(* CODESYS project CORE.library
   Company: Ziga Javornik
   DefaultNamespace: ZigaLibs.Core
   Version: 0.0.3.7
   Placeholder: ZigaLibs.Core
   Author: Ziga Javornik
   Description: A collection of core objects for work with further libraries implementations.
   Title: ZigaLibs.Core

Project tree, tasks and I/O mapping:
  libraries: Base Interfaces, * (System); Tc2_EtherCAT, * (Beckhoff Automation GmbH); Tc2_IoFunctions, 3.4.5.0 (Beckhoff Automation GmbH); Tc2_Standard, * (Beckhoff Automation GmbH); Tc2_System, * (Beckhoff Automation GmbH); Tc2_Utilities, * (Beckhoff Automation GmbH); Tc3_Module, * (Beckhoff Automation GmbH); TcError, 0.2.2.1 (Roald87); TcUnit, * (www.tcunit.org)
  GVLs/
  SOURCE/
    Array/
      DUTs/
        data type ST_ArrayProperties
        data type T_ArrayIndexer
      program ArrayHelper [ST]: Clear, DoesArrayContainItem, FindLastOccupiedItem, GetElementCount, GetMaxIndex, InsertAtStart, SetAtFirstEmptySlot, ShiftDown, ShiftUp, ValidateArrayVar
    Beckhoff/
      Ads/
        program AdsHelper [ST]: GetEthercatMasterIdFromNetIdString, NetIdToString
        function block FB_HasAmsAddressFromProcessImage [ST]: AmsAddress
        interface I_HasAmsAddress: AmsAddress
      EtherCAT/
        CoE/
          DUTs/
            data type ST_CoeEntry
            data type ST_CoeEntry_DINT
            data type ST_CoeEntry_INT
            data type ST_CoeEntry_REAL
            data type ST_CoeEntry_SINT
            data type ST_CoeEntry_String128
            data type ST_CoeEntry_String255
            data type ST_CoeEntry_String30
            data type ST_CoeEntry_UDINT
            data type ST_CoeEntry_UINT
            data type ST_CoeEntry_USINT
            data type T_CoEIndex
            data type T_CoESubIndex
          function block FB_CoeReadWrite [ST]: ReadAny, WriteAny
          interface I_ReadsCoE: ReadCoE
        Diagnosis/
          DUTs/
            Device state/
              data type E_EcDeviceState
              data type E_EcDeviceStateExtras
              data type E_EcLinkState
              data type ST_EcDeviceState
              data type ST_EcSlaveState
            data type E_EthercatDiagnosisState
            data type E_EthercatDiagnosisStatus
            data type ST_EthercatSlaveInfo
          interface I_EthercatDiagnosis: Error, IgnoredSlaves, IgnoreSlave, MissingSlaves, Reset, Scan, Status
        program EthercatHelper [ST]: ConvertBeckhoffEcStateToCustomStruct, GetBoxNameByAddress
        function block FB_ReadBoxName [ST]
    Errors/
      DUTs/
        data type ST_AdsError
        data type ST_Error
        data type ST_GenericError
      function block FB_ErrorSource [ST]: AdsError, Error, GenericError, ResetError
      interface I_ErrorSource
      interface I_HasAdsError: AdsError
      interface I_HasError: Error
      interface I_HasGenericError: GenericError
    General/
      Memory/
        data type E_MemCmpResults
        function block FB_Malloc [ST]: FB_exit, FB_init, ValidateAction, ValidateIndex, ValidateInputVar, IsAllocated, Properties, Allocate, AllocateAny, Expand, Free, Get, GetPtr, Remove, Set
        program MemoryHelper [ST]: GetRouterStatusInfo
        data type ST_AllocatedMemoryProperties
      Variable extensions/
        function block BoolEx [ST]: HasBeenFalseForAtLeast, HasBeenTrueForAtLeast, HasFallingEdge, HasRisingEdge, IsVarValid, PulseWithInterval, Reset, Set, Toggle, Value
      Variable information/
        function F_DoesVarTypeEqual [ST]
        function F_GetVarInfo [ST]
        data type ST_VarInfo
        data type T_VarInfo
        data type T_VarSize
      function block FB_BooleanObserver [ST]
      function block FB_HasInstanceNameAndPath [ST]: FB_init, InstanceName, InstancePath
      function block FB_HasTaskInfo [ST]: TaskInfo
      function block FB_Watchdog [ST]
      program InstanceNameHelper [ST]: InstanceNameFromPath, RemoveProjectFromInstancePath
      data type ST_Value
    String/
      StringBuilder/
        Extensions/
          AddAny/
            data type E_AddAnyBitOptions
            interface I_StringBuilderEx_Any: AddAny, AddAnyBit, AddAnyReal
        function block FB_StringBuilder [ST]: AddAny, AddAnyBit, AddAnyReal, AddString, AddWithDblQuotationMarks, AddWithQuotationMark, Create, Reset
        interface I_StringBuilder: AddString, AddWithDblQuotationMarks, AddWithQuotationMark, Create, Reset
      program StringConstants [ST]
      program StringHelper [ST]: EndsWith, FindStringWithin, Join, StartsWith, ToLowerCase, ToLowerCase_UnlimitedSize, ToUpperCase, ToUpperCase_UnlimitedSize, TrimLeftSide, TrimRightSide
      data type T_Char
    Time/
      DUTs/
        data type E_TimeFormat
        data type ST_CurrentSystemTimeInfo
      function block FB_DateTimeToStringConverter [ST]: DateTime, Day, Hour, Millisecond, Minute, Month, Second, Year
      function block FB_LocalSystemTimeProvider [ST]: ConvertToString, CurrentTime, SetSystemTime
      interface I_DateTimeToStringConverter: DateTime, Day, Hour, Millisecond, Minute, Month, Second, Year
      interface I_LocalSystemTimeProvider: ConvertToString, CurrentTime
  TESTS/
    Test suites/
      Time/
        function block FB_LocalSystemTime_Tests [ST]: Test01_CheckSystemTime_ExpectValue, Test02_SetSystemTime_ExpectNoErrorAndCorrectTimeRead
      function block FB_AdsHelper_Tests [ST]: Test_MasterAddress, Test_NetIdToString_AllZeros_ExpectEmptyString
      function block FB_ArrayHelper_Tests [ST]: Test01_GetArrayElementCount, Test02_GetArrayMaxIndex, Test03_InsertNumber, Test04_InsertString, Test05_InsertStruct, Test06_ShiftUp_ExpectLastElementOverwriteFirstElementZero, Test07_SetAtFirstEmptySlot, Test08_AllMethods_provideNonArrayVar_ExpectNothing, Test09_InsertIntoEmptyArray_ExpectOnlyFirstItem, Test10_CheckIfArrayContainsItem, Test11_ClearArray_ExpectEmptyArray, Test12_ReferenceToArrayWithAllMethods_ExpectNormalResults, Test13_FindLastOccupiedItem, Test14_ShiftDown_ExpectFirstElementOverwriteLastElementZero
      function block FB_BoolEx_Tests [ST]: Test01_BooleanTrue_ExpectTrueAfterElapsedTime, Test02_BooleanFalse_ExpectTrueAfterElapsedTime, Test03_RisingAndFallingEdge_ExpectPulses, Test04_GetAndSetValue, Test05_Toggle_ExpectValueInverts, Test06_PulseWithInterval_100ms_ExpectValueChangeEvery100ms, Test07_Set_ExpectTrue, Test08_Reset_ExpectFalse
      function block FB_DateTimeToStringConverter_Tests [ST]: Test01_Year, Test02_Month, Test03_Day, Test04_Hour, Test05_Minute, Test06_Second, Test07_Millisecond
      function block FB_ErrorSource_ExtensionForTests [ST]
      function block FB_ErrorSource_Tests [ST]: Test01_ErrorProperty, Test02_ErrorCode, Test03_ErrorMessage, Test04_GenericError
      function block FB_EthercatHelper_Tests [ST]: Test01_ConvertBeckhoffEcState_ProvideAllOptions_ExpectCorrectResults
      function block FB_HasInstanceName_ExtensionForTests [ST]
      function block FB_HasInstanceName_Tests [ST]: Test01_InstanceName, Test02_InstancePath
      function block FB_HasTaskInfo_ExtensionsForTests [ST]
      function block FB_HasTaskInfo_Tests [ST]: Test01_TaskInfoPropertyValidity
      function block FB_Malloc_Tests [ST]: BeforeTestFinish, BeforeTestStart, ValidatePropertiesAfterFailedAllocation, Test01_ProvideIncorrectParameters_ExpectNoAllocation, Test02_Allocate10Integers_ExpectNoError_ValidateProperties, Test03_Free_ExpectNoMemoryAllocated, Test04_SetAndGet_ExpectGetReturnsCorrectValue, Test05_SetAtIncorrectIndex_ExpectFalseReturned, Test06_GetFromIncorrectIndex_ExpectTargetValueUnchanged_MethodReturnFalse, Test07_Expand_ExpectOldDataStillExists_LastDataSetIsEmpty, Test08_Remove_ExpectDataSetToCollapseBy1
      function block FB_StringBuilder_Tests [ST]: Test01_AddStrings_ExpectConcat, Test02_AddWithSingleQuotationMarks, Test03_AddWithDoubleQuotationMarks, Test04_CreateDoesNotResetStringSequence, Test05_ResetClearsBuildSequence
      function block FB_StringBuilderEx_Any_Tests [ST]: Test01_BOOL, Test02_BYTE, Test03_DATE, Test04_DateAndTime, Test05_DINT, Test06_DWORD, Test07_ENUM, Test08_INT, Test09_LINT, Test10_LREAL, Test11_LTIME, Test12_LWORD, Test13_REAL, Test14_SINT, Test15_STRING, Test16_TIME, Test17_TOD, Test18_UDINT, Test19_UINT, Test20_ULINT, Test21_USINT, Test22_WORD, Test23_WSTRING, Test24_ANY_BIT_WORD, Test25_ANY_BIT_BYTE, Test26_ANY_BIT_DWORD, Test27_ANY_BIT_LWORD, Test28_ANY_REAL_REAL, Test29_ANY_REAL_LREAL
      function block FB_StringHelper_Tests [ST]: Test01_StartsWith, Test02_Join, Test03_EndsWith, Test05_Contains, Test06_ToLowerCase_UnlimitedSize, Test07_ToUpperCase_UnlimitedSize
    program PRG_TESTS [ST]
*)

// SOURCE/Array/DUTs/ST_ArrayProperties
TYPE ST_ArrayProperties :
STRUCT
	Count		: DINT;
	StartIndex	: T_ArrayIndexer;
	EndIndex	: T_ArrayIndexer;
END_STRUCT
END_TYPE

// SOURCE/Array/DUTs/T_ArrayIndexer
// Should be used when accessing array index.
TYPE T_ArrayIndexer : DINT; END_TYPE

// SOURCE/Beckhoff/EtherCAT/CoE/DUTs/ST_CoeEntry
{attribute 'qualified_only'}
// CoE entry in the dictionary, includes index and the subindex
TYPE ST_CoeEntry :
STRUCT
	Index		: T_CoEIndex;
	Subindex	: T_CoESubIndex;
END_STRUCT
END_TYPE

// SOURCE/Beckhoff/EtherCAT/CoE/DUTs/ST_CoeEntry_DINT
TYPE ST_CoeEntry_DINT EXTENDS ST_CoeEntry :
STRUCT
	Value	: DINT;
END_STRUCT
END_TYPE

// SOURCE/Beckhoff/EtherCAT/CoE/DUTs/ST_CoeEntry_INT
TYPE ST_CoeEntry_INT EXTENDS ST_CoeEntry :
STRUCT
	Value	: INT;
END_STRUCT
END_TYPE

// SOURCE/Beckhoff/EtherCAT/CoE/DUTs/ST_CoeEntry_REAL
TYPE ST_CoeEntry_REAL EXTENDS ST_CoeEntry :
STRUCT
	Value	: REAL;
END_STRUCT
END_TYPE

// SOURCE/Beckhoff/EtherCAT/CoE/DUTs/ST_CoeEntry_SINT
TYPE ST_CoeEntry_SINT EXTENDS ST_CoeEntry :
STRUCT
	Value	: SINT;
END_STRUCT
END_TYPE

// SOURCE/Beckhoff/EtherCAT/CoE/DUTs/ST_CoeEntry_String128
TYPE ST_CoeEntry_String128 EXTENDS ST_CoeEntry :
STRUCT
	Value	: STRING(128);
END_STRUCT
END_TYPE

// SOURCE/Beckhoff/EtherCAT/CoE/DUTs/ST_CoeEntry_String255
TYPE ST_CoeEntry_String255 EXTENDS ST_CoeEntry :
STRUCT
	Value	: Tc2_System.T_MaxString;
END_STRUCT
END_TYPE

// SOURCE/Beckhoff/EtherCAT/CoE/DUTs/ST_CoeEntry_String30
TYPE ST_CoeEntry_String30 EXTENDS ST_CoeEntry :
STRUCT
	Value	: STRING(30);
END_STRUCT
END_TYPE

// SOURCE/Beckhoff/EtherCAT/CoE/DUTs/ST_CoeEntry_UDINT
TYPE ST_CoeEntry_UDINT EXTENDS ST_CoeEntry :
STRUCT
	Value	: UDINT;
END_STRUCT
END_TYPE

// SOURCE/Beckhoff/EtherCAT/CoE/DUTs/ST_CoeEntry_UINT
TYPE ST_CoeEntry_UINT EXTENDS ST_CoeEntry :
STRUCT
	Value	: UINT;
END_STRUCT
END_TYPE

// SOURCE/Beckhoff/EtherCAT/CoE/DUTs/ST_CoeEntry_USINT
TYPE ST_CoeEntry_USINT EXTENDS ST_CoeEntry :
STRUCT
	Value	: USINT;
END_STRUCT
END_TYPE

// SOURCE/Beckhoff/EtherCAT/CoE/DUTs/T_CoEIndex
TYPE T_CoEIndex : WORD; END_TYPE

// SOURCE/Beckhoff/EtherCAT/CoE/DUTs/T_CoESubIndex
TYPE T_CoESubIndex : BYTE; END_TYPE

// SOURCE/Beckhoff/EtherCAT/Diagnosis/DUTs/Device state/E_EcDeviceState
{attribute 'qualified_only'}
TYPE E_EcDeviceState :
(
	INIT		:= Tc2_EtherCAT.EC_DEVICE_STATE_INIT,
	PREOP		:= Tc2_EtherCAT.EC_DEVICE_STATE_PREOP,
	BOOTSTRAP	:= Tc2_EtherCAT.EC_DEVICE_STATE_BOOTSTRAP,
	SAFEOP		:= Tc2_EtherCAT.EC_DEVICE_STATE_SAFEOP,
	OP			:= Tc2_EtherCAT.EC_DEVICE_STATE_OP
)BYTE;
END_TYPE

// SOURCE/Beckhoff/EtherCAT/Diagnosis/DUTs/Device state/E_EcDeviceStateExtras
{attribute 'qualified_only'}
TYPE E_EcDeviceStateExtras :
(
	NOTHING				:= 16#00,
	STATE_MACHINE_ERROR := Tc2_EtherCAT.EC_DEVICE_STATE_ERROR,
	INVALID_VPRS		:= Tc2_EtherCAT.EC_DEVICE_STATE_INVALID_VPRS,
	INIIT_CMD_ERROR		:= Tc2_EtherCAT.EC_DEVICE_STATE_INITCMD_ERROR,
	DISABLED			:= Tc2_EtherCAT.EC_DEVICE_STATE_DISABLED
)BYTE;
END_TYPE

// SOURCE/Beckhoff/EtherCAT/Diagnosis/DUTs/Device state/E_EcLinkState
TYPE E_EcLinkState :
(
	OK					:= Tc2_EtherCAT.EC_LINK_STATE_OK,
	NOT_PRESENT			:= Tc2_EtherCAT.EC_LINK_STATE_NOT_PRESENT,
	LINK_WITHOUT_COMM	:= Tc2_EtherCAT.EC_LINK_STATE_LINK_WITHOUT_COMM,
	MISSING_LINK		:= Tc2_EtherCAT.EC_LINK_STATE_MISSING_LINK,
	ADDITIONAL_LINK		:= Tc2_EtherCAT.EC_LINK_STATE_ADDITIONAL_LINK,
	PORT_A				:= Tc2_EtherCAT.EC_LINK_STATE_PORT_A,
	PORT_B				:= Tc2_EtherCAT.EC_LINK_STATE_PORT_B,
	PORT_C				:= Tc2_EtherCAT.EC_LINK_STATE_PORT_C,
	PORT_D				:= Tc2_EtherCAT.EC_LINK_STATE_PORT_D
)BYTE;
END_TYPE

// SOURCE/Beckhoff/EtherCAT/Diagnosis/DUTs/Device state/ST_EcDeviceState
TYPE ST_EcDeviceState :
STRUCT
	State		: E_EcDeviceState;	// Device state
	StateExtras	: E_EcDeviceStateExtras;	// Extra information
END_STRUCT
END_TYPE

// SOURCE/Beckhoff/EtherCAT/Diagnosis/DUTs/Device state/ST_EcSlaveState
TYPE ST_EcSlaveState :
STRUCT
	Device	: ST_EcDeviceState;	// Device state
	Link	: E_EcLinkState;	// Link state
END_STRUCT
END_TYPE

// SOURCE/Beckhoff/EtherCAT/Diagnosis/DUTs/E_EthercatDiagnosisState
{attribute 'qualified_only'}
{attribute 'strict'}
TYPE E_EthercatDiagnosisState :
(
	READY,
	GET_SLAVE_STATES,
	GET_FAULTY_SLAVE_ADDRESSES,
	FINISHED,
	ERROR
);
END_TYPE

// SOURCE/Beckhoff/EtherCAT/Diagnosis/DUTs/E_EthercatDiagnosisStatus
TYPE E_EthercatDiagnosisStatus :
(
	NO_ERROR,				// No error, all slaves are present
	MISSING_ALLOWED_SLAVES,	// Missing slaves, but they are allowed (for example, hot connect)
	ERROR					// Missing slaves that are not allowed to be missing
);
END_TYPE

// SOURCE/Beckhoff/EtherCAT/Diagnosis/DUTs/ST_EthercatSlaveInfo
TYPE ST_EthercatSlaveInfo :
STRUCT
	Name		: Tc2_System.T_MaxString;	// Slave name
	IsIgnored	: BOOL;	// True if slave is ignored with the scan
	State		: ST_EcSlaveState;
END_STRUCT
END_TYPE

// SOURCE/Errors/DUTs/ST_AdsError
TYPE ST_AdsError EXTENDS ST_Error:
STRUCT
	Code	: TcError.AdsErrorCodes;
	Message	: Tc2_System.T_MaxString;
END_STRUCT
END_TYPE

// SOURCE/Errors/DUTs/ST_Error
TYPE ST_Error :
STRUCT
	Source	: Tc2_System.T_MaxString;
END_STRUCT
END_TYPE

// SOURCE/Errors/DUTs/ST_GenericError
TYPE ST_GenericError EXTENDS ST_Error :
STRUCT
	Code	: DINT;
	Message	: Tc2_System.T_MaxString;
END_STRUCT
END_TYPE

// SOURCE/General/Memory/E_MemCmpResults
{attribute 'qualified_only'}
TYPE E_MemCmpResults :
(
	pBUFF1_LESS_THAN_pBUFF2	:= -1,
	IDENTICAL	:= 0,
	PbUFF1_GREATER_THAN_pBUFF2	:= 1,
	ERROR	:= 255
)DINT;
END_TYPE

// SOURCE/General/Memory/ST_AllocatedMemoryProperties
// Properties for working with dynamic memory allocation.
TYPE ST_AllocatedMemoryProperties :
STRUCT
	Size				: DINT;		// Size of the allocated memory
	StartAddress		: PVOID;	// Pointer to the address of the array memory space
	BaseTypeSize		: DINT;		// Size of the base type provided, when allocated
	NumberOfElements	: DINT;	// Number of elements provided, when allocated.
END_STRUCT
END_TYPE

// SOURCE/General/Variable information/ST_VarInfo
TYPE ST_VarInfo :
STRUCT
	DataType	: __SYSTEM.TYPE_CLASS;
	Address		: POINTER TO BYTE;
	Size		: T_VarSize;
END_STRUCT
END_TYPE

// SOURCE/General/Variable information/T_VarInfo
TYPE T_VarInfo : __SYSTEM.VAR_INFO; END_TYPE

// SOURCE/General/Variable information/T_VarSize
// Variable size alias type. To be used when working with SIZEOF operator.
TYPE T_VarSize : UXINT; END_TYPE

// SOURCE/General/ST_Value
TYPE ST_Value :
STRUCT
	Setpoint	: REAL;
	Actual		: REAL;
END_STRUCT
END_TYPE

// SOURCE/String/StringBuilder/Extensions/AddAny/E_AddAnyBitOptions
{attribute 'qualified_only'}
{attribute 'strict'}
// Provides various options of how ANY_BIT data type can be converted.
TYPE E_AddAnyBitOptions :
(
	BINARY,			// Will be converted to a binary string (base 2)
	DECIMAL,		// Will be converted to a decial string (base 10)
	HEXADECIMAL,	// Will be converted to hexadecimal string (base 16)
	OCTAL			// Will be converted to octal string (base 8)
);
END_TYPE

// SOURCE/String/T_Char
TYPE T_Char : STrING(1); END_TYPE

// SOURCE/Time/DUTs/E_TimeFormat
{attribute 'qualified_only'}
{attribute 'strict'}
TYPE E_TimeFormat :
(
	HHMMSS,
	DDMMYY,
	YYMMDD,
	MMDDYY,
	DDMMYY_HHMMSS,
	YYMMDD_HHMMSS,
	MMDDYY_HHMMSS
);
END_TYPE

// SOURCE/Time/DUTs/ST_CurrentSystemTimeInfo
TYPE ST_CurrentSystemTimeInfo :
STRUCT
	IsValid	: BOOL;
	Value	: Tc2_Utilities.TIMESTRUCT;
END_STRUCT
END_TYPE

// SOURCE/Array/ArrayHelper
{attribute 'enable_dynamic_creation'}
// Provides array helper methods for easier work with arrays accross programming.
PROGRAM ArrayHelper

// Clears the entire array. Returns TRUE if operation was sucessfull.
METHOD PUBLIC Clear : BOOL
VAR_INPUT
	arr			: ANY;	// Array to be cleared
END_VAR
IF NOT ValidateArrayVar(arr) THEN
	RETURN;
END_IF

Tc2_System.MEMSET(
	destAddr := arr.pValue,
	fillByte := 0,
	n := DINT_TO_UDINT(arr.diSize));
	
Clear := TRUE;
END_METHOD

// Looks trough the array and returns TRUE if any element equals to the one provided.
METHOD DoesArrayContainItem : BOOL
VAR_INPUT
	arr		: ANY;	// Array to be checked
	item	: ANY;	// Item to be found in the array
END_VAR

VAR
	itemCount	: T_ArrayIndexer;
	currentItem	: T_ArrayIndexer;
	cmpResult	: E_MemCmpResults;
END_VAR
IF NOT ValidateArrayVar(arr) THEN
	RETURN;
END_IF

IF item.diSize = 0 OR_ELSE	// If item size is 0
	(arr.diSize MOD item.diSize) <> 0 	// If incorrect item is provided (division will return non 0 remainder)
THEN
	RETURN;
END_IF

itemCount := arr.diSize/item.diSize;

FOR currentItem := 0 TO itemCount - 1 BY 1 DO
	cmpResult := Tc2_System.MEMCMP(
		pBuf1 := arr.pValue + DINT_TO_DWORD(currentItem * item.diSize),
		pBuf2 := item.pValue,
		n := DINT_TO_UDINT(item.diSize));
		
	IF cmpResult = E_MemCmpResults.IDENTICAL THEN
		DoesArrayContainItem := TRUE;
		RETURN;
	END_IF
END_FOR
END_METHOD

// Looks trough the array and return the last non-zero element to the result variable.
// Returns TRUE if an element was found and FALSE if no empty elements are found.
// Note that this method uses memmory allocation. All occupied memory is released after method finishes.
METHOD PUBLIC FindLastOccupiedItem	: BOOL
VAR_INPUT
	arr			: ANY;	// Array to look for the last element value
	dataType	: ANY;	// Data type of the array elements, can be used like this : datayType := arr[0]
	result		: ANY;	// Result variable, result be written to this variable
END_VAR

VAR
	i								: T_ArrayIndexer;
	maxIndex						: T_ArrayIndexer;
	compareResult					: E_MemCmpResults;
	ptrAllocatedBytes_emptyElement	: POINTER TO BYTE;
END_VAR
IF NOT ValidateArrayVar(arr) OR result.TypeClass <> dataType.TypeClass THEN
	RETURN;
END_IF

maxIndex :=  GetElementCount(arr := arr, dataType := dataType) - 1;
ptrAllocatedBytes_emptyElement := __NEW(BYTE, DINT_TO_UDINT(dataType.diSize));

// Array with 1 element - loop would point to invalid position, exit early by just checking the values
IF maxIndex = 0 THEN
	IF arr.pValue^ <> ptrAllocatedBytes_emptyElement^ THEN
		Tc2_System.MEMCPY(
			srcAddr := arr.pValue,
			destAddr := result.pValue,
			n := DINT_TO_UDINT(dataType.diSize));
			FindLastOccupiedItem := TRUE;
	END_IF
	// Delete allocated memory and return from the method
	__DELETE(ptrAllocatedBytes_emptyElement);
	RETURN;
END_IF

FOR i := maxIndex TO 0 BY -1 DO
	compareResult := Tc2_System.MEMCMP(
		pBuf1 := arr.pValue +  DINT_TO_DWORD(i * dataType.diSize),
		pBuf2 := ptrAllocatedBytes_emptyElement,
		n := DINT_TO_UDINT(dataType.diSize));
		
	// If element is not empty, return
	IF compareResult <> E_MemCmpResults.IDENTICAL THEN
		Tc2_System.MEMCPY(
			srcAddr := arr.pValue +  DINT_TO_DWORD(i * dataType.diSize),
			destAddr := result.pValue,
			n := DINT_TO_UDINT(dataType.diSize));
		FindLastOccupiedItem := TRUE;
		EXIT;
	END_IF
END_FOR

// Delete allocated memory
__DELETE(ptrAllocatedBytes_emptyElement);
END_METHOD

// Returns the number of elements in the array.
METHOD PUBLIC GetElementCount : DINT
VAR_INPUT
	arr			: ANY;	// Array to be checked.
	dataType	: ANY;	// Data type of the array elements, can be used like this : datayType := arr[0]
END_VAR
IF ValidateArrayVar(arr) = FALSE THEN
	RETURN;
END_IF

IF dataType.diSize = 0 THEN
	RETURN;
END_IF
GetElementCount := arr.diSize / dataType.diSize;
END_METHOD

// Gets the maximum array index that can be used for looping or index accessing
METHOD PUBLIC GetMaxIndex : DINT
VAR_INPUT
	arr			: ANY;	// Array to be checked.
	dataType	: ANY;	// Data type of the array elements, can be used like this : datayType := arr[0]
	startIndex	: T_ArrayIndexer;
END_VAR
IF ValidateArrayVar(arr) = FALSE THEN
	RETURN;
END_IF

GetMaxIndex := startIndex + GetElementCount(arr := arr, dataType := dataType) - 1;
END_METHOD

// Inserts the item to the start of the array. 
// Array contents are shifted by 1, last item is deleted.
METHOD InsertAtStart : BOOL
VAR_INPUT	
	arr		: ANY;	// Array to be checked.
	item	: ANY;	// Item to be inserted on start
 END_VAR
IF ValidateArrayVar(arr) = FALSE THEN
	RETURN;
END_IF

ShiftUp(
	arr := arr,
	dataType := item);

// Set first element value
Tc2_System.MEMCPY(
	destAddr := arr.pValue,
	srcAddr := item.pValue,
	n := DINT_TO_UDINT(item.diSize));
END_METHOD

// Iterates the array and sets the value when first empty slot is found. 
// Note that this method uses memmory allocation. All occupied memory is released after method finishes.
METHOD SetAtFirstEmptySlot
VAR_INPUT
	arr		: ANY;	// Array to be checked.
	item	: ANY;	// Item to set
END_VAR

VAR
	ptrByte 			: POINTER TO BYTE;
	i					: T_ArrayIndexer;
	maxIndex			: T_ArrayIndexer;
	ptrAllocatedBytes	: POINTER TO BYTE;
	cmpResult			: DINT;
END_VAR
IF ValidateArrayVar(arr) = FALSE THEN
	RETURN;
END_IF

maxIndex :=  GetElementCount(arr := arr, dataType := item) - 1;
ptrAllocatedBytes := __NEW(BYTE, DINT_TO_UDINT(arr.diSize));

FOR i := 0 TO maxIndex BY 1 DO
	ptrByte := arr.pValue + DINT_TO_UDINT(item.diSize * i);	
	
	cmpResult := Tc2_System.MEMCMP(
			n := DINT_TO_UDINT(item.diSize),
			pBuf1 := ptrAllocatedBytes,
			pBuf2 := ptrByte);
			
	IF cmpResult = E_MemCmpResults.IDENTICAL THEN
		Tc2_System.MEMCPY(
			destAddr := ptrByte,
			n := DINT_TO_UDINT(item.diSize),
			srcAddr := item.pValue);
		EXIT;
	END_IF
END_FOR

__DELETE(ptrAllocatedBytes);
END_METHOD

// Shifts the array down, losing first element and clearing last element in the process.
METHOD ShiftDown
VAR_INPUT
	arr		: ANY;	// Array to be checked.
	dataType	: ANY;	// Data type of the array elements, can be used like this : datayType := arr[0]
END_VAR
IF ValidateArrayVar(arr) = FALSE THEN
	RETURN;
END_IF

Tc2_System.MEMMOVE(	
	destAddr := arr.pValue,
	srcAddr := arr.pValue + DINT_TO_UDINT(dataType.diSize),
	n := DINT_TO_UDINT(arr.diSize - dataType.diSize));

// Clear last element
Tc2_System.MEMSET(
	fillByte := 0,
	n := DINT_TO_UDINT(dataType.diSize),
	destAddr := arr.pValue + DINT_TO_UDINT(arr.diSize - dataType.diSize));
END_METHOD

// Shifts the array up, losing last element and clearing first element in the process.
METHOD ShiftUp
VAR_INPUT
	arr			: ANY;	// Array to be checked.
	dataType	: ANY;	// Data type of the array elements, can be used like this : datayType := arr[0]
END_VAR
IF ValidateArrayVar(arr) = FALSE THEN
	RETURN;
END_IF


Tc2_System.MEMMOVE(
	destAddr := arr.pValue + DINT_TO_UDINT(dataType.diSize),
	srcAddr := arr.pValue,
	n := DINT_TO_UDINT(arr.diSize - dataType.diSize));

// Clear first element
Tc2_System.MEMSET(
	fillByte := 0,
	n := DINT_TO_UDINT(dataType.diSize),
	destAddr := arr.pValue);
END_METHOD

METHOD PRIVATE ValidateArrayVar : BOOL
VAR_INPUT
	arr	: ANY;
END_VAR
VAR
	isArray		: BOOL;
	isReference	: BOOL;
END_VAR
isArray := F_DoesVarTypeEqual(arr, IBaseLibrary.TYPE_ARRAY);
isReference := F_DoesVarTypeEqual(arr, IBaseLibrary.TYPE_REFERENCE);

ValidateArrayVar := isArray OR isReference;
END_METHOD

END_PROGRAM

// SOURCE/General/Variable information/F_DoesVarTypeEqual
// Returns TRUE if the variable's data type equals to the .
FUNCTION F_DoesVarTypeEqual : BOOL
VAR_INPUT
	variable	: ANY;
	typeClass	: IBaseLibrary.TypeClass;
END_VAR
VAR
END_VAR

F_DoesVarTypeEqual := UDINT_TO_INT(variable.TypeClass) = typeClass;

END_FUNCTION

// SOURCE/Beckhoff/Ads/AdsHelper
// A helper class providing various helpful methods when working with ads data
PROGRAM AdsHelper

// Returns last part of the netId, which is the ID of the etherCAT master.
METHOD PUBLIC GetEthercatMasterIdFromNetIdString : UDINT
VAR_INPUT
	netId	: Tc2_System.T_AmsNetID;
END_VAR

VAR
	sNetIdResult	: T_AmsNetID;
	nMasterAddress	: UDINT;
	nDotPosition	: INT;
END_VAR
sNetIdResult := netId;
nDotPosition := Tc2_Standard.FIND(sNetIdResult, '.');

WHILE nDotPosition <> 0 DO
	nDotPosition := Tc2_Standard.FIND(sNetIdResult, '.');
	IF nDotPosition = 0 THEN
		EXIT;
	END_IF
	sNetIdResult := Tc2_Standard.DELETE(STR := sNetIdResult, POS := 1, LEN := nDotPosition);
END_WHILE

GetEthercatMasterIdFromNetIdString := STRING_TO_UDINT(sNetIdResult);
END_METHOD

// Converts netId of type <Tc2_System.T_AmsNetIdArr> to <T_AmsNetID>, which equates to <STRING(23)>.
METHOD PUBLIC NetIdToString : T_AmsNetID
VAR_INPUT
	netId	: Tc2_System.T_AmsNetIdArr;	// NetId to be converted
END_VAR

VAR
	arrayMaxIndex	: DINT;
	i				: DINT;
END_VAR
arrayMaxIndex := ArrayHelper.GetMaxIndex(
	arr := netId, 
	dataType := netId[0], 
	startIndex := 0);

FOR i := 0 TO arrayMaxIndex BY 1 DO
	// If any element is not 0, exit and call the system function to convert
	IF netId[i] <> 0 THEN
		EXIT;
	END_IF
	// If reaching last element in the array, this means only 0s are present, indicating local netId - return empty string
	IF i = ArrayHelper.GetMaxIndex(arr := netId, dataType := netId[0], startIndex := 0) THEN
		NetIdToString := '';
		RETURN;
	END_IF
END_FOR

NetIdToString := Tc2_System.F_CreateAmsNetId(nIds := netId);
END_METHOD

END_PROGRAM

// SOURCE/Beckhoff/Ads/FB_HasAmsAddressFromProcessImage
// Inherit from this FB to get Tc2_System.ST_AmsAddr in the process image (to link to EtherCAT devices etc...)
FUNCTION_BLOCK ABSTRACT FB_HasAmsAddressFromProcessImage
VAR_INPUT
END_VAR
VAR_OUTPUT
END_VAR
VAR
	Ams AT%I* 	: Tc2_System.ST_AmsAddr;
	_ams 		: Tc2_System.ST_AmsAddr;
END_VAR

(* Gets or sets the Ams address structure*)
PROPERTY AmsAddress : REFERENCE TO Tc2_System.ST_AmsAddr
GET
_ams := Ams;
AmsAddress REF= _ams;
END_GET
END_PROPERTY

END_FUNCTION_BLOCK

// SOURCE/Beckhoff/Ads/I_HasAmsAddress
// Interface to implement when requiring AMS address
INTERFACE I_HasAmsAddress

// Gets or sets the Ams address structure
PROPERTY AmsAddress : REFERENCE TO Tc2_System.ST_AmsAddr
GET
END_GET
SET
END_SET
END_PROPERTY

END_INTERFACE

// SOURCE/Beckhoff/EtherCAT/CoE/FB_CoeReadWrite
FUNCTION_BLOCK FB_CoeReadWrite
VAR
END_VAR

// Reads the CoE parameter at Index:Subindex and writes the value to Value. Returns TRUE when done.
METHOD PUBLIC ReadAny : BOOL
VAR_INPUT
	CoeEntry	: POINTER TO ST_CoeEntry;	// CoE entry, index and subindex
	Value		: ANY;	// Value to where the read result is stored
	SlaveAddr	: AMSADDR;		// Slave AMS address of the device
END_VAR

VAR_INST
	fbCoeRead		: Tc2_EtherCAT.FB_EcCoESdoRead;
	FtrigReadDone	: Tc2_Standard.F_TRIG;
END_VAR
fbCoeRead(
	sNetId:= AdsHelper.NetIdToString(SlaveAddr.netId), 
	nSlaveAddr:= SlaveAddr.port, 
	nSubIndex:= CoeEntry^.Subindex, 
	nIndex:= CoeEntry^.Index, 
	pDstBuf:= Value.pValue, 
	cbBufLen:= DINT_TO_UDINT(Value.diSize), 
	bExecute:= NOT fbCoeRead.bBusy, 
	tTimeout:= T#5S, 
	bError=> , 
	nErrId=> , 
	cbRead=> );

FtrigReadDone(CLK := fbCoeRead.bBusy);
ReadAny := FtrigReadDone.Q;
END_METHOD

// Writes the CoE parameter at Index:Subindex and returns TRUE when done.
METHOD WriteAny : BOOL
VAR_INPUT
	CoeEntry	: POINTER TO ST_CoeEntry;	// CoE entry, index and subindex
	Value		: ANY;	// Value to where the read result is stored
	SlaveAddr	: AMSADDR;		// Slave AMS address of the device
END_VAR

VAR_INST
	fbCoeWrite		: Tc2_EtherCAT.FB_EcCoESdoWrite;
	FtrigWriteDone	: Tc2_Standard.F_TRIG;
END_VAR
fbCoeWrite(
	sNetId:= AdsHelper.NetIdToString(SlaveAddr.netId), 
	nSlaveAddr:= SlaveAddr.port, 
	nSubIndex:= CoeEntry^.Subindex,
	nIndex:= CoeEntry^.Index, 
	pSrcBuf:= Value.pValue, 
	cbBufLen:= DINT_TO_UDINT(Value.diSize), 
	bExecute:= NOT fbCoeWrite.bBusy, 
	tTimeout:= T#3S);
	
FtrigWriteDone(CLK := fbCoeWrite.bBusy, Q => WriteAny);
END_METHOD

END_FUNCTION_BLOCK

// SOURCE/Beckhoff/EtherCAT/CoE/I_ReadsCoE
INTERFACE I_ReadsCoE

// Reads CoE items and updates them. Returns TRUE when done,
// Needs to be called until the method finishes, indicating via the return value. 
METHOD PUBLIC ReadCoE : BOOL
END_METHOD

END_INTERFACE

// SOURCE/Beckhoff/EtherCAT/Diagnosis/I_EthercatDiagnosis
INTERFACE I_EthercatDiagnosis

// Returns TRUE if an error occurred while performing the scan
PROPERTY Error : BOOL
GET
END_GET
END_PROPERTY

// Gets an array of slaves that have been added to ignore list
PROPERTY IgnoredSlaves : REFERENCE TO ARRAY[0..255] OF Tc2_System.T_MaxString
GET
END_GET
END_PROPERTY

// Adds the provided slave to a collection of slaves that will not trigger an error
// Example is slaves that are used on hot connect groups, and when connected should not cause an error. 
METHOD IgnoreSlave
VAR_INPUT
	Name	: Tc2_System.T_MaxString;	// Slave to be ignored if not found or an error is reported back
END_VAR
END_METHOD

// Returns an array of misisng slave names
PROPERTY MissingSlaves : REFERENCE TO ARRAY[0..255] OF ST_EthercatSlaveInfo
GET
END_GET
END_PROPERTY

// Reset the internal state machine of diagnosis and clearing any errors, if active.
METHOD Reset
END_METHOD

// Performs a scan on the EtherCAT master, returns TRUE when done.
METHOD Scan	: BOOL
VAR_INPUT
	EcMasterNetId	: AMSNETID;
END_VAR
END_METHOD

// Gets the status based on last executed scan.
PROPERTY Status : E_EthercatDiagnosisStatus
GET
END_GET
END_PROPERTY

END_INTERFACE

// SOURCE/Beckhoff/EtherCAT/EthercatHelper
{attribute 'hide_all_locals'}
PROGRAM EthercatHelper
VAR
	fbReadDeviceName	: Tc2_IoFunctions.IOF_GetBoxNameByAddr;
	nMasterId			: UDINT;
END_VAR

// Converts Tc2_EtherCAT.ST_EcSlaveState to ZigaLibs_Core.ST_EcSlaveState and returns the converted structure.
METHOD ConvertBeckhoffEcStateToCustomStruct : ST_EcSlaveState
VAR_INPUT
	ecSlaveState	: Tc2_EtherCAT.ST_EcSlaveState;
END_VAR
VAR CONSTANT
	SLAVE_STATE_MASK 		: BYTE := 16#0F;
	SLAVE_STATE_EXTRAS_MASK : BYTE := 16#F0;
END_VAR
ConvertBeckhoffEcStateToCustomStruct.Device.State := SLAVE_STATE_MASK AND ecSlaveState.deviceState;
ConvertBeckhoffEcStateToCustomStruct.Device.StateExtras := SLAVE_STATE_EXTRAS_MASK AND ecSlaveState.deviceState;
ConvertBeckhoffEcStateToCustomStruct.Link := ecSlaveState.linkState;
END_METHOD

METHOD PUBLIC GetBoxNameByAddress : T_MaxString
VAR_INPUT
	PlcRuntimeNetId		: Tc2_System.T_AmsNetID; // NetId of the PLC where the devuce is located
	AmsNetId			: AMSADDR; // NetId of the box
	outError			: REFERENCE TO BOOL;	// If an error occurs while executing, method will provide the error flag here. This is a pointer to YOUR boolean error variable.
END_VAR

VAR
	sNetId	: Tc2_System.T_AmsNetID;
END_VAR
sNetId := AdsHelper.NetIdToString(AmsNetId.netId);
fbReadDeviceName(
	NETID := PlcRuntimeNetId,
	DEVICEID := AdsHelper.GetEthercatMasterIdFromNetIdString(netId := sNetId),
	BOXADDR := AmsNetId.port,
	START := NOT fbReadDeviceName.BUSY);
	
outError := fbReadDeviceName.ERR;
GetBoxNameByAddress := fbReadDeviceName.BOXNAME;
END_METHOD

END_PROGRAM

// SOURCE/Beckhoff/EtherCAT/FB_ReadBoxName
// Reads box name and return string
FUNCTION_BLOCK FB_ReadBoxName
VAR_INPUT
	PlcRuntimeNetId		: Tc2_System.T_AmsNetID; // NetId of the PLC where the devuce is located
	AmsNetId			: AMSADDR; // NetId of the box
END_VAR
VAR_OUTPUT
		error 	:  BOOL;	// If an error occurs while executing, method will provide the error flag here. This is a pointer to YOUR boolean error variable.
		done		: BOOL;
		name		: Tc2_System.T_MaxString;
END_VAR

VAR
	fbReadDeviceName	: Tc2_IoFunctions.IOF_GetBoxNameByAddr;
END_VAR

fbReadDeviceName(
	NETID := PlcRuntimeNetId,
	DEVICEID := AdsHelper.GetEthercatMasterIdFromNetIdString(AdsHelper.NetIdToString(AmsNetId.netId)),
	BOXADDR := AmsNetId.port,
	START := NOT fbReadDeviceName.BUSY);
	
error := fbReadDeviceName.ERR;
name := fbReadDeviceName.BOXNAME;

END_FUNCTION_BLOCK

// SOURCE/Errors/FB_ErrorSource
// Provides I_ErrorSource base implementation.

{attribute 'no_explicit_call' := 'Body contains no logic, calling methods only allowed.'}
FUNCTION_BLOCK ABSTRACT FB_ErrorSource EXTENDS FB_HasInstanceNameAndPath IMPLEMENTS I_ErrorSource
VAR
	_adsError		: ST_AdsError;
	_error			: BOOL;
	_genericError	: ST_GenericError;
END_VAR

// Gets or sets the Ads error - note that code to message conversion is done automatically.
{attribute 'monitoring':='call'}
PROPERTY AdsError : REFERENCE TO ST_AdsError
GET
_adsError.Message := TcError.AdsErrorCodeDescription(_adsError.Code);
AdsError REF= _adsError;
END_GET
SET
PROTECTED 
VAR
END_VAR
_adsError := AdsError;
END_SET
END_PROPERTY

{attribute 'monitoring':='call'}
(* Returns TRUE if an error has occurred*)
PROPERTY Error : BOOL
GET
Error := _error;
END_GET
SET
PROTECTED 
VAR
END_VAR
_error := Error;
END_SET
END_PROPERTY

{attribute 'monitoring':='call'}
PROPERTY GenericError : REFERENCE TO ST_GenericError
GET
GenericError REF= _genericError;
END_GET
SET
PROTECTED 
VAR
END_VAR
_genericError := GenericError;
END_SET
END_PROPERTY

// Reset all errors
METHOD PROTECTED ResetError : BOOL
VAR_INPUT
END_VAR
THIS^.Error := FALSE;
THIS^.AdsError.Code := TcError.ToAdsErrorCode(0);
THIS^.AdsError.Source := '';
THIS^.GenericError.Code := 0;
THIS^.GenericError.Source := '';
END_METHOD

END_FUNCTION_BLOCK

// SOURCE/Errors/I_ErrorSource
INTERFACE I_ErrorSource EXTENDS I_HasAdsError, I_HasGenericError, I_HasError

END_INTERFACE

// SOURCE/Errors/I_HasAdsError
INTERFACE I_HasAdsError

{attribute 'monitoring':='call'}
// Gets or sets the Ads error - note that code to message conversion is done automatically.
PROPERTY AdsError : REFERENCE TO ST_AdsError
GET
END_GET
END_PROPERTY

END_INTERFACE

// SOURCE/Errors/I_HasGenericError
INTERFACE I_HasGenericError

{attribute 'monitoring':='call'}
// Gets the Generic error
PROPERTY GenericError : REFERENCE TO ST_GenericError
GET
END_GET
END_PROPERTY

END_INTERFACE

// SOURCE/Errors/I_HasError
INTERFACE I_HasError

{attribute 'monitoring':='call'}
// Returns TRUE if an error has occurred
PROPERTY Error : BOOL
GET
END_GET
END_PROPERTY

END_INTERFACE

// SOURCE/General/FB_HasInstanceNameAndPath
// When inherited, the child function block will gain two properties:
// InstanceName - ONLY the name of the instantiated function block
// InstancePath - the FULL instance path

{attribute 'reflection'}
{attribute 'hide_all_locals'}
{attribute 'no_explicit_call' := 'Body contains no logic, calling methods only allowed.'}
FUNCTION_BLOCK ABSTRACT FB_HasInstanceNameAndPath
VAR
	{attribute 'instance-path'} 
    {attribute 'noinit'} 
	_instancePath	: Tc2_System.T_MaxString;
	_instanceName	: Tc2_System.T_MaxString;
END_VAR

{attribute 'hide'}
METHOD FB_init : BOOL
VAR_INPUT
	bInitRetains : BOOL; // if TRUE, the retain variables are initialized (warm start / cold start)
	bInCopyCode : BOOL;  // if TRUE, the instance afterwards gets moved into the copy code (online change)
END_VAR
_instanceName := InstanceNameHelper.InstanceNameFromPath(_instancePath, 10);
_instancePath := InstanceNameHelper.RemoveProjectFromInstancePath(_instancePath);
END_METHOD

{attribute 'monitoring':='call'}
PROPERTY InstanceName : Tc2_System.T_MaxString
GET
InstanceName := _instanceName;
END_GET
END_PROPERTY

{attribute 'monitoring':='call'}
PROPERTY InstancePath : Tc2_System.T_MaxString
GET
VAR
	varInfo	: T_VarInfo;
END_VAR
InstancePath := _instancePath;
END_GET
END_PROPERTY

END_FUNCTION_BLOCK

// SOURCE/General/InstanceNameHelper
PROGRAM InstanceNameHelper
VAR
END_VAR

METHOD InstanceNameFromPath : T_MaxString
VAR_INPUT
	path		: Tc2_System.T_MaxString;
	maxAttempts	: INT;
END_VAR
VAR
	instanceName	: Tc2_System.T_MaxString;
	dotPosition		: INT;
	iteration		: INT;
	
END_VAR

VAR CONSTANT
	ABSOLUTE_MAX_ATTEMPTS : INT := 20;
END_VAR
instanceName := path;

// Limiting maximum number of dots in the instancePath to maximum of 20 with ABSOLUTE_MAX_ATTEMPTS
// This is mostly important due to the method being called in FB_Init, where I think too long method calls shouldn't be happening.
// In theory, I don't think it would ever go above 10, unless some very deep object nesting is done.
// Example Project.Plc.Main.Fb.Fb.Fb.Fb.Fb...

WHILE Tc2_Standard.FIND(STR1 := instanceName, STR2 := '.') <> 0 AND 
	 (iteration < MIN(maxAttempts, ABSOLUTE_MAX_ATTEMPTS)) 
DO
	dotPosition := Tc2_Standard.FIND(
		STR1 := instanceName, 
		STR2 := '.');
		
	instanceName := Tc2_Standard.DELETE(
		STR := instanceName,
		POS := 1,	
		LEN := dotPosition);
		
	iteration := iteration + 1;
END_WHILE

InstanceNameFromPath := instanceName;
END_METHOD

METHOD RemoveProjectFromInstancePath : T_MaxString
VAR_INPUT
	instancePath	: Tc2_System.T_MaxString;
END_VAR
VAR
	result		: Tc2_System.T_MaxString;
	dotPosition	: INT;
	iteration	: INT;
END_VAR

VAR CONSTANT
	FILE_PREIX_DOTS_TO_REMOVE	: INT := 2;
END_VAR
RemoveProjectFromInstancePath := InstanceNameFromPath(instancePath,2);
END_METHOD

END_PROGRAM

// SOURCE/General/Memory/FB_Malloc
{attribute 'enable_dynamic_creation'}
// Function block for memory allocation. It only handles a single memory instance.
FUNCTION_BLOCK FB_Malloc
VAR
	_allocated	: POINTER TO BYTE;
	_properties	: ST_AllocatedMemoryProperties;
END_VAR

METHOD FB_exit : BOOL
VAR_INPUT
	bInCopyCode : BOOL; // if TRUE, the exit method is called for exiting an instance that is copied afterwards (online change).
END_VAR
Free();
END_METHOD

METHOD FB_init : BOOL
VAR_INPUT
	bInitRetains : BOOL; // if TRUE, the retain variables are initialized (warm start / cold start)
	bInCopyCode : BOOL;  // if TRUE, the instance afterwards gets moved into the copy code (online change)
	baseTypeSize	: DINT;	// Base data type's that will be used
	elementCount	: DINT;	// Number of elements
END_VAR
Allocate(baseTypeSize, elementCount);
END_METHOD

METHOD PRIVATE ValidateAction : BOOL
VAR_INPUT
	index		: DINT;
	variable	: ANY;
END_VAR
ValidateAction := ValidateIndex(index) AND ValidateInputVar(variable) AND IsAllocated;
END_METHOD

METHOD PRIVATE ValidateIndex : BOOL
VAR_INPUT
	index	: DINT;
END_VAR
ValidateIndex := index <= (_properties.NumberOfElements - 1) AND index >= 0;
END_METHOD

METHOD PRIVATE ValidateInputVar : BOOL
VAR_INPUT
	variable	: ANY;
END_VAR
ValidateInputVar := variable.diSize = _properties.BaseTypeSize;
END_METHOD

{attribute 'monitoring':='call'}
// Returns TRUE if memory has been allocated.
PROPERTY PUBLIC IsAllocated : BOOL
GET
IsAllocated := _properties.StartAddress  <> 0;
END_GET
END_PROPERTY

{attribute 'monitoring':='call'}
// Gets properties of the allocated memory.
PROPERTY Properties : REFERENCE TO ST_AllocatedMemoryProperties
GET
Properties REF= _properties;
END_GET
END_PROPERTY

// Allocates the memory of size = elementSize * numberOfElements.
// If the memory allocation has already been done, Free() will be called first!
// Returns TRUE if allocation has been sucessfull - this can fail if incorrect parameters are provided (sie <= 0 or numberOfElements = 0)
METHOD Allocate : BOOL
VAR_INPUT
	elementSize			: DINT;	// Size of the element.
	numberOfElements	: DINT;	// Number of elements that will occupy the memory space.
END_VAR
IF elementSize <= 0 OR numberOfElements <= 0 THEN
	RETURN;
END_IF

Free();
_allocated := __NEW(BYTE, DINT_TO_UDINT((elementSize * numberOfElements)));

_properties.BaseTypeSize := elementSize;
_properties.NumberOfElements := numberOfElements;
_properties.Size := elementSize * numberOfElements;
_properties.StartAddress := _allocated;

Allocate := _allocated <> 0;
END_METHOD

// Allocates memory based on the provided parameters
// If the memory allocation has already been done, Free() will be called first!
METHOD AllocateAny : BOOL
VAR_INPUT
	dataType			: ANY;		// Provide the variable that will be used as base type here
	numberOfElements	: DINT;	// Number of elements that should be allocated.
END_VAR
AllocateAny :=  Allocate(dataType.diSize, numberOfElements);
END_METHOD

// Expands the current allocated memory
METHOD Expand : BOOL
VAR_INPUT
	elementsToAdd	: DINT; // Number of new elements to be added. Only accepting values larger than 0.
END_VAR
VAR
	oldAllocatedMemory	: POINTER TO BYTE;
	originalProperties	: ST_AllocatedMemoryProperties;
END_VAR
IF NOT IsAllocated OR elementsToAdd <= 0 THEN
	RETURN;
END_IF

// Copy current contents
originalProperties := _properties;
oldAllocatedMemory := __NEW(BYTE, (DINT_TO_UDINT(_properties.Size)));

Tc2_System.MEMCPY(
	srcAddr := _allocated, 
	destAddr := oldAllocatedMemory,
 	n := DINT_TO_UDINT(_properties.Size));

// Free the memory	
THIS^.Free();

// Create new, expanded memory
THIS^.Allocate(
	elementSize := originalProperties.BaseTypeSize ,
	numberOfElements:=  originalProperties.NumberOfElements + elementsToAdd);
	
// Copy the old values to the new allocation.	
Tc2_System.MEMCPY(
	srcAddr := oldAllocatedMemory,
	destAddr := _allocated,
	n := DINT_TO_UDINT(originalProperties.Size));
	
// Delete the temporary allocated memory
__DELETE(oldAllocatedMemory);
END_METHOD

// Frees the allocated memory area. 
// Returns TRUE if operation was executed (if nothing is allocated, then FALSE is returned).
METHOD Free : BOOL
VAR_INPUT
END_VAR
IF _allocated <> 0 THEN
	__DELETE(_allocated);
	_properties.BaseTypeSize := 0;
	_properties.NumberOfElements := 0;
	_properties.Size := 0;
	_properties.StartAddress := 0;
	Free := TRUE;
	RETURN;
END_IF
END_METHOD

// Gets the value at the provided 'index' copies it to the 'result' variable.
METHOD Get : BOOL
VAR_INPUT
	index	: DINT;
	result	: ANY;
END_VAR
IF NOT ValidateAction(index,result) THEN
	Get := FALSE;
	RETURN;
END_IF

Tc2_System.MEMCPY(
	destAddr := result.pValue,	
	srcAddr := _properties.StartAddress + DINT_TO_UDINT(index * _properties.BaseTypeSize),
	n := DINT_TO_UDINT(_properties.BaseTypeSize));
	
Get := TRUE;
END_METHOD

// Gets the pointer to the provided index
// This can be used to alter the contents by using POINTER TO <DATA_TYPE>. by calling it from another method
METHOD GetPtr : PVOID
VAR_INPUT
	index	: DINT;
END_VAR
IF THIS^.ValidateIndex(index) AND 
   THIS^.IsAllocated 
THEN
	GetPtr := _properties.StartAddress + DINT_TO_UDINT(index * _properties.BaseTypeSize);
END_IF
END_METHOD

// Removes the element at the index.
METHOD Remove	: BOOL;
VAR_INPUT
	index	: DINT;
END_VAR

VAR
	byteCountLowerPart	: DINT;
	byteCountUpperPart	: DINT;
	upperPart			: POINTER TO BYTE;
	lowerPart			: POINTER TO BYTE;
	originalProperties	: ST_AllocatedMemoryProperties;
	newSize				: DINT;
	combinedSize		: DINT;
END_VAR
IF NOT IsAllocated OR NOT ValidateIndex(index) THEN
	RETURN;
END_IF

// If 0th element is the only element, then just free the memory space.
IF index = 0 AND _properties.NumberOfElements = 1 THEN
	Remove := TRUE;
	THIS^.Free();
	RETURN;
END_IF

originalProperties := _properties;
byteCountLowerPart := _properties.BaseTypeSize * index;
lowerPart := __NEW(BYTE, DINT_TO_UDINT(byteCountLowerPart));
Tc2_System.MEMCPY(
	srcAddr := _allocated,
	destAddr := lowerPart,
	n := DINT_TO_UDINT(byteCountLowerPart));
	
byteCountUpperPart := _properties.BaseTypeSize * (_properties.NumberOfElements - 1 - index );
IF byteCountUpperPart <> 0 THEN
	upperPart := __NEW(BYTE, DINT_TO_UDINT(byteCountUpperPart));
	Tc2_System.MEMCPY(
		srcAddr := _allocated + DINT_TO_DWORD(_properties.Size) -  DINT_TO_DWORD(byteCountUpperPart),
		destAddr := upperPart,
		n := DINT_TO_UDINT(byteCountUpperPart));	
END_IF

THIS^.Free();

// For debug purpose, new size and combined size should be the same.
newSize := originalProperties.NumberOfElements - 1;
combinedSize := (byteCountLowerPart + byteCountUpperPart) / originalProperties.BaseTypeSize;

THIS^.Allocate(originalProperties.BaseTypeSize, newSize);
Tc2_System.MEMCPY(
	srcAddr := lowerPart,
	destAddr := _allocated,
	n := DINT_TO_UDINT(byteCountLowerPart));
	
IF byteCountUpperPart <> 0 THEN
	Tc2_System.MEMCPY(
		srcAddr := upperPart,
		destAddr := _allocated + DINT_TO_UDINT(byteCountLowerPart),
		n := DINT_TO_UDINT(byteCountUpperPart));
END_IF	
	
__DELETE(lowerPart);	
IF upperPart <> 0 THEN
	__DELETE(upperPart);
END_IF

Remove := TRUE;
END_METHOD

METHOD Set : BOOL
VAR_INPUT
	index	: DINT;
	value	: ANY;
END_VAR
IF NOT ValidateAction(index,value) THEN
	Set := FALSE;
	RETURN;
END_IF

Tc2_System.MEMCPY(
	destAddr := _properties.StartAddress + DINT_TO_UDINT(index * _properties.BaseTypeSize),	
	srcAddr := value.pValue,
	n := DINT_TO_UDINT(_properties.BaseTypeSize));
	
Set := TRUE;
END_METHOD

END_FUNCTION_BLOCK

// SOURCE/General/Memory/MemoryHelper
{attribute 'hide_all_locals'}
PROGRAM MemoryHelper

VAR
	_getRouterStatusInfo : Tc2_Utilities.FB_GetRouterStatusInfo;
END_VAR

// Gets the router info and copies it to the refRouterInfo. Returns TRUE when done.
METHOD GetRouterStatusInfo : BOOL
VAR_INPUT
	netId			: Tc2_System.T_AmsNetID;
	refRouterInfo	: REFERENCE TO Tc2_Utilities.ST_TcRouterStatusInfo;
END_VAR

VAR_INST
	
END_VAR
_getRouterStatusInfo(
	bExecute := NOT _getRouterStatusInfo.bBusy,
	sNetId := netId);
	
refRouterInfo := _getRouterStatusInfo.info;
GetRouterStatusInfo := NOT _getRouterStatusInfo.bBusy;
END_METHOD

END_PROGRAM

// SOURCE/General/Variable extensions/BoolEx
// An extension to boolean variable
FUNCTION_BLOCK BoolEx
VAR_INPUT
	variable			: REFERENCE TO BOOL;
END_VAR

VAR
	
	_risingEdge			: Tc2_Standard.R_TRIG;
	_fallingEdge		: Tc2_Standard.F_TRIG;
	afterinitvarinfo 	: ST_VarInfo;
END_VAR

// Returns TRUE if monitored value has been FALSE for at lease for the provided "duration"
METHOD HasBeenFalseForAtLeast : BOOL
VAR_INPUT
	duration	: TIME;
END_VAR

VAR_INST
	timer	: Tc2_Standard.TON;

END_VAR
IF NOT IsVarValid() THEN
	RETURN;
END_IF

timer(IN := NOT variable, PT := duration);
HasBeenFalseForAtLeast := timer.Q;
END_METHOD

// Returns TRUE if monitored value has been TRUE for at lease for the provided "duration"
METHOD HasBeenTrueForAtLeast : BOOL
VAR_INPUT
	duration	: TIME;
END_VAR

VAR_INST
	timer	: Tc2_Standard.TON;
	ptrBool	: POINTER TO BOOL;
END_VAR
IF NOT IsVarValid() THEN
	RETURN;
END_IF

timer(IN := variable, PT := duration);
HasBeenTrueForAtLeast := timer.Q;
END_METHOD

// Returns TRUE if oberved variable change from TRUE to FALSE from the last call.
PROPERTY HasFallingEdge : BOOL
GET
_fallingEdge(CLK := variable);
HasFallingEdge := _fallingEdge.Q;
END_GET
END_PROPERTY

// Returns TRUE if oberved variable change from FALSE to TRUE from the last call.
PROPERTY HasRisingEdge : BOOL
GET
_risingEdge(CLK := variable);
HasRisingEdge := _risingEdge.Q;
END_GET
END_PROPERTY

METHOD PROTECTED IsVarValid : BOOL
IsVarValid := __ISVALIDREF(variable);
END_METHOD

// Pulses the virabile (TRUE/FALSE) with the provided on and off duration
METHOD PulseWithInterval
VAR_INPUT
	durationOn	: TIME;
	durationOff	: TIME;
END_VAR
VAR_INST
	timerOn		: Tc2_Standard.TON;
	timerOff	: Tc2_Standard.TON;
END_VAR
IF NOT IsVarValid() THEN
	RETURN;
END_IF
// In order to properly trigger immediate change, call both timers twice. 
// This way when ON is elapsed, OFF starts imediately and vice versa.
timerOff(IN := timerOn.Q, PT := durationOff);
timerOn(IN := NOT timerOff.Q, PT := durationOn);
timerOff(IN := timerOn.Q, PT := durationOff);
timerOn(IN := NOT timerOff.Q, PT := durationOn);
variable := NOT timerOn.Q;
END_METHOD

// Sets the value to FALSE
METHOD Reset
VAR_INPUT
END_VAR
IF NOT IsVarValid() THEN
	RETURN;
END_IF

variable := FALSE;
END_METHOD

// Sets the value to TRUE
METHOD Set
VAR_INPUT
END_VAR
IF NOT IsVarValid() THEN
	RETURN;
END_IF

variable := TRUE;
END_METHOD

METHOD Toggle
IF NOT IsVarValid() THEN
	RETURN;
END_IF

variable := NOT variable;
END_METHOD

PROPERTY Value : BOOL
GET
Value := variable;
END_GET
SET
variable := Value;
END_SET
END_PROPERTY

END_FUNCTION_BLOCK

// SOURCE/General/Variable information/F_GetVarInfo
// Returns information about the variable as ST_VarInfo.
FUNCTION F_GetVarInfo : ST_VarInfo
VAR_INPUT
	variable	: ANY;	// Variable to get the inforation from
END_VAR
VAR
END_VAR

F_GetVarInfo.Address := variable.pValue;
F_GetVarInfo.DataType := variable.TypeClass;
F_GetVarInfo.Size := DINT_TO_UDINT(variable.diSize);

END_FUNCTION

// SOURCE/General/FB_BooleanObserver
// Boolean condition observer. Body requires calling every cycle in order to execute the triggers!
// Checkes the "bCondition" and returns a 1 cycle pulse output on bRisingEdge when value changes form 0 to 1
// Checkes the "bCondition" and returns a 1 cycle pulse output on bFallingEdge when value changes form 1 to 0

FUNCTION_BLOCK FB_BooleanObserver
VAR_INPUT
	bCondition	: BOOL;
END_VAR
VAR_OUTPUT
	bRisingEdge		: BOOL;
	bFallingEdge	: BOOL;
END_VAR
VAR
	_rtrig	: Tc2_Standard.R_TRIG;
	_ftrig	: Tc2_Standard.F_TRIG;
END_VAR

_rtrig(CLK := bCondition, Q => bRisingEdge);
_ftrig(CLK := bCondition, Q => bFallingEdge);

END_FUNCTION_BLOCK

// SOURCE/General/FB_HasTaskInfo
{attribute 'no_explicit_call' := 'Body contains no logic, calling methods only allowed.'}
FUNCTION_BLOCK ABSTRACT FB_HasTaskInfo
VAR
	_PlcTaskInfo	: REFERENCE TO PlcTaskSystemInfo;
END_VAR

{attribute 'monitoring':='call'}
PROPERTY TaskInfo : REFERENCE TO PlcTaskSystemInfo
GET
VAR
	taskIndex	: DINT;
END_VAR
IF NOT __ISVALIDREF(_plcTaskInfo) OR_ELSE _plcTaskInfo.CycleTime = 0 THEN
	taskIndex := Tc2_System.GETCURTASKINDEXEX();
	IF taskIndex <> 0 THEN
		_PlcTaskInfo REF= TwinCAT_SystemInfoVarList._TaskInfo[taskIndex];
	END_IF
END_IF

TaskInfo REF= _PlcTaskInfo;
END_GET
END_PROPERTY

END_FUNCTION_BLOCK

// SOURCE/General/FB_Watchdog
// A watchdog function block. Observer "variable" input - if the value does not change within the "timeout" parameter, status will return "FALSE"
FUNCTION_BLOCK FB_Watchdog
VAR_INPUT
	variable	: BOOL;	// Variable to observe
	timeout		: TIME;	// Time within the variable needs to change it's state before status is reported as FALSE
END_VAR

VAR_OUTPUT
	status	: BOOL;	// TRUE = OK, FALSE = timeout
END_VAR

VAR
	Ton_TrueTimer	: Tc2_Standard.TON;
	Ton_Falsetimer	: Tc2_Standard.TON;
END_VAR

Ton_TrueTimer(IN := variable, PT := timeout);
Ton_Falsetimer(IN := NOT variable, PT := timeout);


status := Ton_TrueTimer.Q = FALSE AND  Ton_Falsetimer.Q = FALSE;

END_FUNCTION_BLOCK

// SOURCE/String/StringBuilder/Extensions/AddAny/I_StringBuilderEx_Any
INTERFACE I_StringBuilderEx_Any

(* Adds the variable of any data type to the sequence. Conversion is done automatically from within.
Some extra info: 
	- BOOL and BIT will have the string converted to 'TRUE' and 'FALSE' respectively.
	- floating point variables will have their values precision based on constructor realFormatPrecision and will be rounded based on the roundRealValues
*)
METHOD AddAny : REFERENCE TO FB_StringBuilder
VAR_INPUT
	anyVar	: ANY;
END_VAR
END_METHOD

// Adds a variable of type ANY_BIT to the string generating sequence, based on the provided parameters.
// This includes: BYTE, WORD, DWORD, LWORD, 
METHOD AddAnyBit : REFERENCE TO FB_StringBuilder
VAR_INPUT
	anyBit					: ANY_BIT;				// Value to be converterd
	option					: E_AddAnyBitOptions;	// Select how the value is converter
	lowerCase				: BOOL;					// If hexadecimal option is selected, the result string can be converted to either lower or upper case
	displayedDigitsCount	: INT;					// This determines how many digits are to be displayed. If actual digits count is lower, the string is filled with zeros from the left side. If left at 0, the result string will be an empty string!
	addNotation				: BOOL;					// If this is set to TRUE, a notation will be prepended: (DEC)10, (BIN)10, (HEX)10, (OCT)10
END_VAR
END_METHOD

// Adds any REAL or LREAL value to the generating string sequence.
// Please note that REAL values will ALWAYS be automatically rounded on 3rd decimal digit.
// Anything after it will be whatever TwinCAT representation decides to do.
METHOD AddAnyReal : REFERENCE TO FB_StringBuilder
VAR_INPUT
	anyReal		: ANY_REAL;	// Value to be converter
	precision	: INT;		// Precision
	round		: BOOL;		// Rounding of the last displayed digit
END_VAR
END_METHOD

END_INTERFACE

// SOURCE/String/StringBuilder/FB_StringBuilder
(* Provides basic string builder implementation.
IMPORTANT NOTE! Doing too many method chains might cause the codesys compiler to either be very slow
when doing the "generating code" part or even fail. Restrain to not using too many or too
many nested methods ( method(fb.Method(fb2.Method())... ).
*)
FUNCTION_BLOCK FB_StringBuilder IMPLEMENTS I_StringBuilder, I_StringBuilderEx_Any 
VAR
	_string	: Tc2_System.T_MaxString;
END_VAR

(* Adds the variable of any data type to the sequence. Conversion is done automatically from within. 
Returns I_StringBuilderEx_Any for further string building capability.

Some extra info: 
	- BOOL and BIT will have the string converted to 'TRUE' and 'FALSE' respectively.
	- BYTE, WORD, DWORD and LWORD will be converted without any additional options. Use AddAnyBit method for these instead!
	- REAL and LREAL will be added as T_MaxString values. Please use AddAnyReal method for these instead.*)

METHOD AddAny : REFERENCE TO FB_StringBuilder
VAR_INPUT
	anyVar	: ANY;
END_VAR

VAR
	result	: Tc2_System.T_MaxString;
	ptrWstring	: POINTER TO WSTRING;
END_VAR
CASE TO_INT(anyVar.TypeClass) OF 
	IBaseLibrary.TypeClass.TYPE_BOOL:
		IF Tc2_Utilities.PBOOL_TO_BOOL(anyVar.pValue) = TRUE THEN
			result :=	'TRUE';
		ELSE
			result := 'FALSE';
		END_IF
		
	IBaseLibrary.TypeClass.TYPE_BYTE: 
		result := BYTE_TO_STRING(Tc2_Utilities.PBYTE_TO_BYTE(anyVar.pValue));
	
	IBaseLibrary.TypeClass.TYPE_DATE:
		result := DATE_TO_STRING(Tc2_Utilities.PDATE_TO_DATE(anyVar.pValue));
	
	IBaseLibrary.TypeClass.TYPE_DATEANDTIME:
		result := DT_TO_STRING(Tc2_Utilities.PDT_TO_DT(anyVar.pValue));
	
	IBaseLibrary.TypeClass.TYPE_DINT:
		result := DINT_TO_STRING(Tc2_Utilities.PDINT_TO_DINT(anyVar.pValue));
	
	IBaseLibrary.TypeClass.TYPE_DWORD:
		result := DWORD_TO_STRING(Tc2_Utilities.PDWORD_TO_DWORD(anyVar.pValue));
	
	IBaseLibrary.TypeClass.TYPE_ENUM:
		result := TO_STRING(anyVar.pValue^);
	
	IBaseLibrary.TypeClass.TYPE_INT:
		result := INT_TO_STRING(Tc2_Utilities.PINT_TO_INT(anyVar.pValue));
	
	IBaseLibrary.TypeClass.TYPE_LINT:
		result := LINT_TO_STRING(Tc2_Utilities.PLINT_TO_LINT(anyVar.pValue));
		
	IBaseLibrary.TypeClass.TYPE_LREAL:
		result := LREAL_TO_STRING(Tc2_Utilities.PLREAL_TO_LREAL(anyVar.pValue));
	
	IBaseLibrary.TypeClass.TYPE_LTIME:
		result := LTIME_TO_STRING(Tc2_Utilities.PLTIME_TO_LTIME(anyVar.pValue));
		
	IBaseLibrary.TypeClass.TYPE_LWORD:
		result := LWORD_TO_STRING(Tc2_Utilities.PLWORD_TO_LWORD(anyVar.pValue));
		
	IBaseLibrary.TypeClass.TYPE_REAL:
		result := REAL_TO_STRING(Tc2_Utilities.PREAL_TO_REAL(anyVar.pValue));
	
	IBaseLibrary.TypeClass.TYPE_SINT:
		result := SINT_TO_STRING(Tc2_Utilities.PSINT_TO_SINT(anyVar.pValue));
	
	IBaseLibrary.TypeClass.TYPE_STRING:
		result := TO_STRING(Tc2_Utilities.PSTRING_TO_STRING(anyVar.pValue));
		
	IBaseLibrary.TypeClass.TYPE_TIME:
		result := TIME_TO_STRING(Tc2_Utilities.PTIME_TO_TIME(anyVar.pValue));
	
	IBaseLibrary.TypeClass.TYPE_TIMEOFDAY:
		result := TOD_TO_STRING(Tc2_Utilities.PTOD_TO_TOD(anyVar.pValue));
	
	IBaseLibrary.TypeClass.TYPE_UDINT:
		result := UDINT_TO_STRING(Tc2_Utilities.PUDINT_TO_UDINT(anyVar.pValue));		
	
	IBaseLibrary.TypeClass.TYPE_UINT:
		result := UINT_TO_STRING(Tc2_Utilities.PUINT_TO_UINT(anyVar.pValue));
	
	IBaseLibrary.TypeClass.TYPE_ULINT:
		result := ULINT_TO_STRING(Tc2_Utilities.PULINT_TO_ULINT(anyVar.pValue));
	
	IBaseLibrary.TypeClass.TYPE_USINT:
		result := USINT_TO_STRING(Tc2_Utilities.PUSINT_TO_USINT(anyVar.pValue));
	
	IBaseLibrary.TypeClass.TYPE_WORD:
		result := WORD_TO_STRING(Tc2_Utilities.PWORD_TO_WORD(anyVar.pValue));
	
	IBaseLibrary.TypeClass.TYPE_WSTRING:
		ptrWstring := anyVar.pValue;
		result := WSTRING_TO_STRING(ptrWstring^);
		
	ELSE
		result := TO_STRING(anyVar.pValue^);
	
END_CASE

THIS^.AddString(result);
AddAny REF= THIS^;
END_METHOD

// Adds a variable of type ANY_BIT to the string generating sequence, based on the provided parameters.
// This includes: BYTE, WORD, DWORD, LWORD, 
METHOD AddAnyBit  : REFERENCE TO FB_StringBuilder
VAR_INPUT
	anyBit					: ANY_BIT;				// Value to be converterd
	option					: E_AddAnyBitOptions;	// Select how the value is converter
	lowerCase				: BOOL;					// If hexadecimal option is selected, the result string can be converted to either lower or upper case
	displayedDigitsCount	: INT;					// This determines how many digits are to be displayed. If actual digits count is lower, the string is filled with zeros from the left side. If left at 0, the result string will be an empty string!
	addNotation				: BOOL;					// If this is set to TRUE, a notation will be prepended: (DEC)10, (BIN)10, (HEX)10, (OCT)10
END_VAR
VAR
	result : Tc2_System.T_MaxString;
END_VAR
CASE anyBit.TypeClass OF
	__SYSTEM.TYPE_CLASS.TYPE_WORD:
		CASE option OF
			E_AddAnyBitOptions.BINARY:
				result := Tc2_Utilities.WORD_TO_BINSTR(
					in := anyBit.pValue^,
					iPrecision := displayedDigitsCount);
				
			E_AddAnyBitOptions.DECIMAL:
				result := Tc2_Utilities.WORD_TO_DECSTR(
					in := anyBit.pValue^,
					iPrecision := displayedDigitsCount);
				
			E_AddAnyBitOptions.HEXADECIMAL:
				result := Tc2_Utilities.WORD_TO_HEXSTR(
					in := anyBit.pValue^,
					iPrecision := displayedDigitsCount,
					bLoCase := lowerCase);
				
			E_AddAnyBitOptions.OCTAL:
				result := Tc2_Utilities.WORD_TO_OCTSTR(
					in := anyBit.pValue^,
					iPrecision := displayedDigitsCount);
		END_CASE
		
	__SYSTEM.TYPE_CLASS.TYPE_BYTE:
		CASE option OF
			E_AddAnyBitOptions.BINARY:
				result := Tc2_Utilities.BYTE_TO_BINSTR(
					in := anyBit.pValue^,
					iPrecision := displayedDigitsCount);
				
			E_AddAnyBitOptions.DECIMAL:
				result := Tc2_Utilities.BYTE_TO_DECSTR(
					in := anyBit.pValue^,
					iPrecision := displayedDigitsCount);
				
			E_AddAnyBitOptions.HEXADECIMAL:
				result := Tc2_Utilities.BYTE_TO_HEXSTR(
					in := anyBit.pValue^,
					iPrecision := displayedDigitsCount,
					bLoCase := lowerCase);
				
			E_AddAnyBitOptions.OCTAL:
				result := Tc2_Utilities.BYTE_TO_OCTSTR(
					in := anyBit.pValue^, 
					iPrecision := displayedDigitsCount);
		END_CASE
	
	__SYSTEM.TYPE_CLASS.TYPE_DWORD:
		CASE option OF
			E_AddAnyBitOptions.BINARY:
				result := Tc2_Utilities.WORD_TO_BINSTR(
					in := anyBit.pValue^,
					iPrecision := displayedDigitsCount);
				
			E_AddAnyBitOptions.DECIMAL:
				result := Tc2_Utilities.WORD_TO_DECSTR(
					in := anyBit.pValue^,
					iPrecision := displayedDigitsCount);
				
			E_AddAnyBitOptions.HEXADECIMAL:
				result := Tc2_Utilities.WORD_TO_HEXSTR(
					in := anyBit.pValue^,
					iPrecision := displayedDigitsCount,
					bLoCase := lowerCase);
				
			E_AddAnyBitOptions.OCTAL:
				result := Tc2_Utilities.WORD_TO_OCTSTR(
					in := anyBit.pValue^,
					iPrecision := displayedDigitsCount);
		END_CASE
	
	__SYSTEM.TYPE_CLASS.TYPE_LWORD:
		CASE option OF
			E_AddAnyBitOptions.BINARY:
				result := Tc2_Utilities.LWORD_TO_BINSTR(
					in := anyBit.pValue^,
					iPrecision := displayedDigitsCount);
				
			E_AddAnyBitOptions.DECIMAL:
				result := Tc2_Utilities.LWORD_TO_DECSTR(
					in := anyBit.pValue^,
					iPrecision := displayedDigitsCount);
				
			E_AddAnyBitOptions.HEXADECIMAL:
				result := Tc2_Utilities.LWORD_TO_HEXSTR(
					in := anyBit.pValue^,
					iPrecision := displayedDigitsCount,
					bLoCase := lowerCase);
				
			E_AddAnyBitOptions.OCTAL:
				result := Tc2_Utilities.LWORD_TO_OCTSTR(
					in := anyBit.pValue^,
					iPrecision := displayedDigitsCount);
		END_CASE
END_CASE

IF addNotation THEN
	CASE option OF
		E_AddAnyBitOptions.BINARY:
			result := Tc2_Standard.CONCAT('(BIN)', result);
			
		E_AddAnyBitOptions.DECIMAL:
			result := Tc2_Standard.CONCAT('(DEC)', result);
		
		E_AddAnyBitOptions.HEXADECIMAL:
			result := Tc2_Standard.CONCAT('(HEX)', result);
		
		E_AddAnyBitOptions.OCTAL:
			result := Tc2_Standard.CONCAT('(OCT)', result);
	END_CASE
END_IF

THIS^.AddString(result);
AddAnyBit REF= THIS^;
END_METHOD

// Adds any REAL or LREAL value to the generating string sequence.
// Please note that REAL values will ALWAYS be automatically rounded on 3rd decimal digit.
// Anything after it will be whatever TwinCAT decides to do.
METHOD AddAnyReal : REFERENCE TO FB_StringBuilder
VAR_INPUT
	anyReal		: ANY_REAL;	// Value to be converter
	precision	: INT;		// Precision of decimal digits
	round		: BOOL;		// Rounding of the last displayed digit
END_VAR
IF anyReal.diSize = SIZEOF(REAL) THEN
	// REAL
	THIS^.AddString(
		Tc2_Utilities.LREAL_TO_FMTSTR(
			in := REAL_TO_LREAL(Tc2_Utilities.PREAL_TO_REAL(anyReal.pValue)),
			iPrecision := precision, 
			bRound := round));
		
ELSE
	// LREAL
	THIS^.AddString(Tc2_Utilities.LREAL_TO_FMTSTR(
		in := Tc2_Utilities.PLREAL_TO_LREAL(anyReal.pValue),
		iPrecision := precision,
		bRound := round));	
END_IF

AddAnyReal REF= THIS^;
END_METHOD

(* Adds a string to the build sequence.*)
METHOD AddString : REFERENCE TO FB_StringBuilder
VAR_INPUT
	(* String to be added.*)
	str	: Tc2_System.T_MaxString;
END_VAR
_string := Tc2_Standard.CONCAT(
	STR1 := _string, 
	STR2 := str);
	
AddString  REF= THIS^;
END_METHOD

(* Adds a string to the build sequence and wraps the str in double quotation marks "str"*)
METHOD AddWithDblQuotationMarks : REFERENCE TO FB_StringBuilder
VAR_INPUT
	str	: Tc2_System.T_MaxString;
END_VAR
_string := Tc2_Standard.CONCAT(
	STR1 := _string, 
	STR2 := Tc2_Standard.CONCAT(
		STR1 := StringConstants.DoubleQuotationMark, 
		STR2 := Tc2_Standard.CONCAT(
			STR1 := str, 
			STR2 := StringConstants.DoubleQuotationMark))); 
	
AddWithDblQuotationMarks  REF= THIS^;
END_METHOD

(* Adds a string to the build sequence and wraps the str in quotation marks 'str'*)
METHOD AddWithQuotationMark : REFERENCE TO FB_StringBuilder
VAR_INPUT
	str	: Tc2_System.T_MaxString;
END_VAR
_string := Tc2_Standard.CONCAT(
	STR1 := _string, 
	STR2 := Tc2_Standard.CONCAT(
		STR1 := StringConstants.SingleQuotationMark, 
		STR2 := Tc2_Standard.CONCAT(
			STR1 := str, 
			STR2 := StringConstants.SingleQuotationMark))); 
		
AddWithQuotationMark REF= THIS^;
END_METHOD

(* Finishes string generation and returns the generated string*)
METHOD Create : Tc2_System.T_MaxString
Create := _string;
END_METHOD

(* Reset the string build sequence, clear any string built so far.*)
METHOD Reset : REFERENCE TO FB_StringBuilder
_string := '';
Reset REF= THIS^;
END_METHOD

END_FUNCTION_BLOCK

// SOURCE/String/StringBuilder/I_StringBuilder
INTERFACE I_StringBuilder

// Adds a string to the build sequence.
METHOD AddString : REFERENCE TO FB_StringBuilder
VAR_INPUT
	str	: Tc2_System.T_MaxString;	// String to be added.
END_VAR
END_METHOD

// Adds a string to the build sequence and wraps the str in double quotation marks "str"
METHOD AddWithDblQuotationMarks : REFERENCE TO FB_StringBuilder
VAR_INPUT
	str : Tc2_System.T_MaxString;
END_VAR
END_METHOD

// Adds a string to the build sequence and wraps the str in quotation marks 'str'
METHOD AddWithQuotationMark : REFERENCE TO FB_StringBuilder
VAR_INPUT
	str	: Tc2_System.T_MaxString;
END_VAR
END_METHOD

// Finishes string generation and returns the generated string
METHOD Create : Tc2_System.T_MaxString
END_METHOD

(* Reset the string build sequence, clear any string built so far.*)
METHOD Reset : REFERENCE TO FB_StringBuilder
VAR_INPUT
END_VAR
END_METHOD

END_INTERFACE

// SOURCE/String/StringConstants
(* Contains string constants
A STRING constant is a string enclosed by single quotation marks. The characters are encoded according to the Windows 1252 character set. 
As a subset of Windows-1252, the character set of ISO/IEC 8859-1 is supported. 
A STRING constant can contain blanks and umlauts, since these characters are part of the character set. 
It is also referred to as a character literal or simply a string.*)

PROGRAM StringConstants
VAR CONSTANT
	LineFeed			: STRING := '$L';
	NewLine				: STRING := '$N';
	FormFeed			: STRING := '$P';
	LineBreak			: STRING := '$R';
	Tab					: STRING := '$T';
	DollarSign			: STRING := '$$';
	SingleQuotationMark	: STRING := '$'';
	DoubleQuotationMark	: STRING := '$22';
END_VAR

END_PROGRAM

// SOURCE/String/StringHelper
PROGRAM StringHelper
VAR
END_VAR

METHOD EndsWith : BOOL
VAR_INPUT
	str		: Tc2_System.T_MaxString;
	char	: T_Char;	
END_VAR
EndsWith := Tc2_Standard.RIGHT(str, 1) = char;
END_METHOD

// Checks if the sourceString contains the stringToFind string. 
// Size of the source string is only limited to TwinCAT limitaitons, which in theory is not limited.
// Returns TRUE if found, else FALSE. Position of the found strimg is provided in the "position" output variable.
METHOD FindStringWithin : BOOL
VAR_INPUT
	sourceString	: ANY;	// String to look at
	stringToFind	: Tc2_System.T_MaxString; // String that should be containted in the sourceString
END_VAR
VAR_OUTPUT
	position	: DINT;	// Position of the found string
END_VAR

VAR
	tmpStr						: POINTER TO Tc2_System.T_MaxString;
	charIndex					: DINT;
	currentMatchingCharIndex	: DINT;
	tmpByte						: POINTER TO BYTE;
	firstCharPosition 			: dint;
END_VAR
IF NOT F_DoesVarTypeEqual(sourceString, IBaseLibrary.TYPE_STRING) THEN
	RETURN;
END_IF

IF sourceString.diSize <= SIZEOF(Tc2_System.T_MaxString) THEN
	tmpStr := __NEW(BYTE, SIZEOF(Tc2_System.T_MaxString));
	Tc2_System.MEMCPY(
		destAddr := tmpStr,
		srcAddr := sourceString.pValue,
		n := DINT_TO_UDINT(sourceString.diSize));
	//tmpStr := sourceString.pValue;
	position :=  Tc2_Standard.FIND(tmpStr^, stringToFind);
	FindStringWithin := position <> 0;
	__DELETE(tmpStr);
	RETURN;
END_IF

FOR charIndex := 0 TO sourceString.diSize BY 1 DO
	
	// Byte wise comparison, if matching byte, start filling the compared string
	tmpByte := sourceString.pValue + charIndex * SIZEOF(BYTE);
	// For debug purpose
	tmpStr := tmpByte;
	IF tmpbyte^ = stringToFind[currentMatchingCharIndex] THEN
		IF firstCharPosition = 0 THEN
			firstCharPosition := charIndex + 1;
		END_IF
		currentMatchingCharIndex := currentMatchingCharIndex + 1;
	ELSE
		currentMatchingCharIndex := 0;
		firstCharPosition := 0;
	END_IF
	
	// When index = str lenght - 1, we have found the entire string, exit the loop.
	IF currentMatchingCharIndex = (Tc2_Standard.LEN(stringToFind)) THEN
		position := firstCharPosition;
		FindStringWithin := TRUE;
		EXIT;
	END_IF
END_FOR
END_METHOD

// Joins the provided string with the string to add.
// The refStr is altered in the process, this no additional assignments are required as oposed to CONCAT which returns the resulting string.
METHOD Join
VAR_INPUT
	refStr		: REFERENCE TO Tc2_System.T_MaxString;
	strToJoin	: Tc2_System.T_MaxString;
END_VAR
refStr := Tc2_Standard.CONCAT(refStr, strToJoin);
END_METHOD

// Checks if STRING `str` starts with the `char`
// Returs TRUE if first character in the provided string is `char` provided
METHOD StartsWith : BOOL
VAR_INPUT
	str		: Tc2_System.T_MaxString;	// String to be checked
	char	: T_Char;	// Character that the string will be checked, if it starts with it.
END_VAR
StartsWith := Tc2_System.F_ToCHR(str[0]) = char;
END_METHOD

// Converts the provided string to all lower case and returns the converted value.
METHOD ToLowerCase : T_MaxString
VAR_INPUT
	str	: Tc2_System.T_MaxString;	// Source string
END_VAR
ToLowerCase := Tc2_Utilities.F_ToLCase(in := str);
END_METHOD

// Converts the input string to all lower case. Size of the string is irrelevant
METHOD ToLowerCase_UnlimitedSize
VAR_INPUT
	str	: ANY;
END_VAR

VAR
	charIndex	: DINT;
	ptrChar		: POINTER TO T_Char;
	char		: T_Char;
	malloc		: FB_Malloc(0,0);
	ptrByte		: POINTER TO BYTE;
END_VAR
IF NOT F_DoesVarTypeEqual(str, IBaseLibrary.TYPE_STRING) THEN
	RETURN;
END_IF

malloc.Allocate(1, str.diSize - 1);		
FOR charIndex := 0 TO str.diSize - 1 BY 1 DO
	ptrChar := str.pValue + DINT_TO_DWORD(charIndex);
	char := ToLowerCase(ptrChar^);
	ptrByte := ADR(char);
	malloc.Set(charIndex, ptrByte^);
END_FOR

Tc2_System.MEMCPY(
	destAddr := str.pValue, 
	srcAddr := malloc.Properties.StartAddress, 
	n := DINT_TO_UDINT(str.diSize - 1));
	
malloc.Free();
END_METHOD

// Converts the provided string to all upper case and returns the converted value.
METHOD ToUpperCase : Tc2_System.T_MaxString
VAR_INPUT
	str	: Tc2_System.T_MaxString;	// Source string
END_VAR
ToUpperCase := Tc2_Utilities.F_ToUCase(in := str);
END_METHOD

METHOD ToUpperCase_UnlimitedSize
VAR_INPUT
	str	: ANY;
END_VAR	

VAR
	charIndex	: DINT;
	ptrChar		: POINTER TO T_Char;
	char		: T_Char;
	malloc		: FB_Malloc(0,0);
	ptrByte		: POINTER TO BYTE;
END_VAR
IF NOT F_DoesVarTypeEqual(str, IBaseLibrary.TYPE_STRING) THEN
	RETURN;
END_IF

malloc.Allocate(1, str.diSize - 1);		
FOR charIndex := 0 TO str.diSize - 1 BY 1 DO
	ptrChar := str.pValue + DINT_TO_DWORD(charIndex);
	char := ToUpperCase(ptrChar^);
	ptrByte := ADR(char);
	malloc.Set(charIndex, ptrByte^);
END_FOR

Tc2_System.MEMCPY(
	destAddr := str.pValue, 
	srcAddr := malloc.Properties.StartAddress, 
	n := DINT_TO_UDINT(str.diSize - 1));
	
malloc.Free();
END_METHOD

// Removes leading spaces from the character string and returns the reduced character string
METHOD PUBLIC TrimLeftSide : Tc2_System.T_MaxString
VAR_INPUT
	str	: Tc2_System.T_MaxString; // String to be trimmed
END_VAR
TrimLeftSide := Tc2_Utilities.F_LTrim(in := str);
END_METHOD

// Truncates all trailing spaces from the specified value and returns the result.
METHOD PUBLIC TrimRightSide : Tc2_System.T_MaxString
VAR_INPUT
	str	: Tc2_System.T_MaxString;	// String to be trimmed
END_VAR
TrimRightSide := Tc2_Utilities.F_RTrim(in := str);
END_METHOD

END_PROGRAM

// SOURCE/Time/FB_DateTimeToStringConverter
FUNCTION_BLOCK FB_DateTimeToStringConverter IMPLEMENTS I_DateTimeToStringConverter
VAR
	_stringBuilder		: FB_StringBuilder;
END_VAR
VAR_IN_OUT
	localSystemTime	: Tc2_Utilities.FB_LocalSystemTime;
END_VAR

(* Converts TIMESTRUCT to STRING.*)
METHOD DateTime : STRING
VAR_INPUT
	timeFormat			: E_TimeFormat;	// Time format to apply to the timestruct conversion
	timeOfDaySeperator	: STRING(1);	// Specifies how time of day is split
	dateSeperator		: STRING(1);	// Specifies how date is split
	fillWithZeros		: BOOL;	// If set to true: month, day hour, minute and second will have 0 added when only a single digit is present
	IncludeMilliseconds	: BOOL; // If set to true, milliseconds will also be displayed in the result, else they are ignored
END_VAR

VAR
	result			: Tc2_System.T_MaxString;
	stringBuilder	: FB_StringBuilder;
END_VAR
{warning disable C0371}

IF NOT __ISVALIDREF(localSystemTime) THEN
	RETURN;
END_IF

CASE timeFormat OF
	E_TimeFormat.DDMMYY:
		result := stringBuilder.Reset()
			.AddString(THIS^.Day(fillWithZeros))
			.AddString(dateSeperator)
			.AddString(THIS^.Month(fillWithZeros))
			.AddString(dateSeperator)
			.AddString(THIS^.Year())
			.Create();

	E_TimeFormat.HHMMSS:
		result := stringBuilder.Reset()
			.AddString(THIS^.Hour(fillWithZeros))
			.AddString(timeOfDaySeperator)
			.AddString(THIS^.Minute(fillWithZeros))
			.AddString(timeOfDaySeperator)
			.AddString(THIS^.Second(fillWithZeros))
			.Create();
			
		IF IncludeMilliseconds THEN
			result := stringBuilder.AddString(timeOfDaySeperator)
				.AddString(THIS^.Millisecond(fillWithZeros))
				.Create();
		END_IF
			
	E_TimeFormat.MMDDYY:
		result := stringBuilder.Reset()
			.AddString(THIS^.Month(fillWithZeros))
			.AddString(dateSeperator)
			.AddString(THIS^.Day(fillWithZeros))
			.AddString(dateSeperator)
			.AddString(THIS^.Year())
			.Create();

	E_TimeFormat.YYMMDD:	
		result := stringBuilder.Reset()
			.AddString(THIS^.Month(fillWithZeros))
			.AddString(dateSeperator)
			.AddString(THIS^.Day(fillWithZeros))
			.AddString(dateSeperator)
			.AddString(THIS^.Year())
			.Create();
		
	E_TimeFormat.DDMMYY_HHMMSS:
		result := stringBuilder.Reset()
			.AddString(THIS^.Day(fillWithZeros))
			.AddString(dateSeperator)
			.AddString(THIS^.Month(fillWithZeros))
			.AddString(dateSeperator)
			.AddString(THIS^.Year())
			.AddString('_')
			.AddString(THIS^.Hour(fillWithZeros))
			.AddString(timeOfDaySeperator)
			.AddString(THIS^.Minute(fillWithZeros))
			.AddString(timeOfDaySeperator)
			.AddString(THIS^.Second(fillWithZeros))
			.Create();
			
			IF IncludeMilliseconds THEN
				result := stringBuilder.AddString(timeOfDaySeperator)
					.AddString(THIS^.Millisecond(fillWithZeros))
					.Create();
			END_IF

	E_TimeFormat.MMDDYY_HHMMSS:
		result := stringBuilder.Reset()
			.AddString(THIS^.Month(fillWithZeros))
			.AddString(dateSeperator)
			.AddString(THIS^.Day(fillWithZeros))
			.AddString(dateSeperator)
			.AddString(THIS^.Year())
			.AddString('_')
			.AddString(THIS^.Hour(fillWithZeros))
			.AddString(timeOfDaySeperator)
			.AddString(THIS^.Minute(fillWithZeros))
			.AddString(timeOfDaySeperator)
			.AddString(THIS^.Second(fillWithZeros))
			.Create();
			
			IF IncludeMilliseconds THEN
				result := stringBuilder.AddString(timeOfDaySeperator)
					.AddString(THIS^.Millisecond(fillWithZeros))
					.Create();
			END_IF

	E_TimeFormat.YYMMDD_HHMMSS:
		result := stringBuilder.Reset()
			.AddString(THIS^.Year())
			.AddString(dateSeperator)
			.AddString(THIS^.Month(fillWithZeros))
			.AddString(dateSeperator)
			.AddString(THIS^.Day(fillWithZeros))
			.AddString('_')
			.AddString(THIS^.Hour(fillWithZeros))
			.AddString(timeOfDaySeperator)
			.AddString(THIS^.Minute(fillWithZeros))
			.AddString(timeOfDaySeperator)
			.AddString(THIS^.Second(fillWithZeros))
			.Create();
			
			IF IncludeMilliseconds THEN
				result := stringBuilder.AddString(timeOfDaySeperator)
					.AddString(THIS^.Millisecond(fillWithZeros))
					.Create();
			END_IF				
END_CASE

DateTime := result;

{warning restore C0371}
END_METHOD

(* Converts TIMESTRUCT.wDay to STRING.*)
METHOD Day : STRING
VAR_INPUT
	fillWithZeros	: BOOL;	// If set to true, result will have 0 added when only a single digit is present
END_VAR
VAR
	result	: STRING;
END_VAR
{warning disable C0371}

IF NOT __ISVALIDREF(localSystemTime) THEN
	RETURN;
END_IF

result := WORD_TO_STRING(localSystemTime.systemTime.wDay);

IF NOT fillWithZeros THEN
	Day := result;
	RETURN;
END_IF

IF Tc2_Standard.LEN(STR := result) < 2 THEN
	result := Tc2_Standard.CONCAT(STR1 := '0', STR2 := result);
END_IF

Day := result;

{warning restore C0371}
END_METHOD

(* Converts TIMESTRUCT.wHour to STRING.*)
METHOD Hour : STRING
VAR_INPUT
	fillWithZeros	: BOOL;	// If set to true, result will have 0 added when only a single digit is present
END_VAR
VAR
	result	: STRING;
END_VAR
{warning disable C0371}

IF NOT __ISVALIDREF(localSystemTime) THEN
	RETURN;
END_IF

result := WORD_TO_STRING(localSystemTime.systemTime.wHour);

IF NOT fillWithZeros THEN
	Hour := result;
	RETURN;
END_IF

IF Tc2_Standard.LEN(STR := result) < 2 THEN
	result := Tc2_Standard.CONCAT(STR1 := '0', STR2 := result);
END_IF

Hour := result;

{warning restore C0371}
END_METHOD

(* Converts TIMESTRUCT.wMillisecond to STRING.*)
METHOD Millisecond : STRING
VAR_INPUT
	fillWithZeros	: BOOL;	// If set to true, result will have 0 added when only a single digit is present
END_VAR
VAR
	result	: STRING;
END_VAR
{warning disable C0371}

IF NOT __ISVALIDREF(localSystemTime) THEN
	RETURN;
END_IF

result := WORD_TO_STRING(localSystemTime.systemTime.wMilliseconds);

IF NOT fillWithZeros THEN
	Millisecond := result;
	RETURN;
END_IF

IF Tc2_Standard.LEN(STR := result) < 3 THEN
	// _10 => 010
	result := Tc2_Standard.CONCAT(STR1 := '0', STR2 := result);
ELSIF Tc2_Standard.LEN(STR := result) < 2 THEN
	// __5 => 005
	result := Tc2_Standard.CONCAT(STR1 := '00', STR2 := result);
END_IF

Millisecond := result;

{warning restore C0371}
END_METHOD

(* Converts TIMESTRUCT.wMinute to STRING.*)
METHOD Minute : STRING
VAR_INPUT
	fillWithZeros	: BOOL;	// If set to true, result will have 0 added when only a single digit is present
END_VAR
VAR
	result	: STRING;
END_VAR
{warning disable C0371}

IF NOT __ISVALIDREF(localSystemTime) THEN
	RETURN;
END_IF

result := WORD_TO_STRING(localSystemTime.systemTime.wMinute);

IF NOT fillWithZeros THEN
	Minute := result;
	RETURN;
END_IF

IF Tc2_Standard.LEN(STR := result) < 2 THEN
	result := Tc2_Standard.CONCAT(STR1 := '0', STR2 := result);
END_IF

Minute := result;

{warning restore C0371}
END_METHOD

(* Converts TIMESTRUCT.wMonth to STRING.*)
METHOD Month : STRING
VAR_INPUT
	fillWithZeros	: BOOL;	// If set to true, result will have 0 added when only a single digit is present
END_VAR
VAR
	result	: STRING;
END_VAR
{warning disable C0371}

IF NOT __ISVALIDREF(localSystemTime) THEN
	RETURN;
END_IF

result := WORD_TO_STRING(localSystemTime.systemTime.wMonth);

IF NOT fillWithZeros THEN
	Month := result;
	RETURN;
END_IF

IF Tc2_Standard.LEN(STR := result) < 2 THEN
	result := Tc2_Standard.CONCAT(STR1 := '0', STR2 := result);
END_IF

Month := result;

{warning restore C0371}
END_METHOD

(* Converts TIMESTRUCT.wSecond to STRING.*)
METHOD Second : STRING
VAR_INPUT
	fillWithZeros	: BOOL;	// If set to true, result will have 0 added when only a single digit is present
END_VAR
VAR
	result	: STRING;
END_VAR
{warning disable C0371}

IF NOT __ISVALIDREF(localSystemTime) THEN
	RETURN;
END_IF

result := WORD_TO_STRING(localSystemTime.systemTime.wSecond);

IF NOT fillWithZeros THEN
	Second := result;
	RETURN;
END_IF

IF Tc2_Standard.LEN(STR := result) < 2 THEN
	result := Tc2_Standard.CONCAT(STR1 := '0', STR2 := result);
END_IF

Second := result;

{warning restore C0371}
END_METHOD

(* Converts TIMESTRUCT.wYear to STRING.*)
METHOD Year : STRING
VAR
	result	: STRING;
END_VAR
{warning disable C0371}

IF NOT __ISVALIDREF(localSystemTime) THEN
	RETURN;
END_IF

result := WORD_TO_STRING(localSystemTime.systemTime.wYear);
Year := result;

{warning restore C0371}
END_METHOD

END_FUNCTION_BLOCK

// SOURCE/Time/I_DateTimeToStringConverter
INTERFACE I_DateTimeToStringConverter

(* Converts TIMESTRUCT to STRING.*)
METHOD DateTime : STRING
VAR_INPUT
	timeFormat			: E_TimeFormat;	// Time format to apply to the timestruct conversion
	timeOfDaySeperator	: STRING(1);	// Specifies how time of day is split
	dateSeperator		: STRING(1);	// Specifies how date is split
	fillWithZeros		: BOOL;	// If set to true: month, day hour, minute and second will have 0 added when only a single digit is present
	IncludeMilliseconds	: BOOL; // If set to true, milliseconds will also be displayed in the result, else they are ignored
END_VAR
END_METHOD

(* Converts TIMESTRUCT.wDay to STRING.*)
METHOD Day : STRING
VAR_INPUT
	fillWithZeros	: BOOL;	// If set to true, result will have 0 added when only a single digit is present
END_VAR
END_METHOD

(* Converts TIMESTRUCT.wHour to STRING.*)
METHOD Hour : STRING
VAR_INPUT
	fillWithZeros	: BOOL;	// If set to true, result will have 0 added when only a single digit is present
END_VAR
END_METHOD

(* Converts TIMESTRUCT.wMillisecond to STRING.*)
METHOD Millisecond : STRING
VAR_INPUT
	fillWithZeros	: BOOL;	// If set to true, result will have 0 added when only a single digit is present
END_VAR
END_METHOD

(* Converts TIMESTRUCT.wMinute to STRING.*)
METHOD Minute : STRING
VAR_INPUT
	fillWithZeros	: BOOL;	// If set to true, result will have 0 added when only a single digit is present
END_VAR
END_METHOD

(* Converts TIMESTRUCT.wMonth to STRING.*)
METHOD Month : STRING
VAR_INPUT
	fillWithZeros	: BOOL;	// If set to true, result will have 0 added when only a single digit is present
END_VAR
END_METHOD

(* Converts TIMESTRUCT.wSecond to STRING.*)
METHOD Second : STRING
VAR_INPUT
	fillWithZeros	: BOOL;	// If set to true, result will have 0 added when only a single digit is present
END_VAR
END_METHOD

(* Converts TIMESTRUCT.wYear to STRING.*)
METHOD Year : STRING
END_METHOD

END_INTERFACE

// SOURCE/Time/FB_LocalSystemTimeProvider
FUNCTION_BLOCK FB_LocalSystemTimeProvider IMPLEMENTS I_LocalSystemTimeProvider
VAR
	_localSystemTime			: Tc2_Utilities.FB_LocalSystemTime;
	_currentSystemTimeInfo		: ST_CurrentSystemTimeInfo;
	_dateTimeToStringCovnerter	: FB_DateTimeToStringConverter;
	_iDateTimeToStringConverter	: I_DateTimeToStringConverter := _dateTimeToStringCovnerter;
END_VAR

_localSystemTime(
	sNetID:= '', 
	bEnable:= TRUE, 
	dwCycle:= 1, 
	systemTime=> _currentSystemTimeInfo.Value);
	
_currentSystemTimeInfo.IsValid := _currentSystemTimeInfo.Value.wYear > 1970;
	
_dateTimeToStringCovnerter(
	localSystemTime := _localSystemTime);

METHOD PUBLIC ConvertToString : I_DateTimeToStringConverter
VAR_INPUT
END_VAR
ConvertToString := _iDateTimeToStringConverter;
END_METHOD

{attribute 'monitoring':='call'}
// Gets current system timo info as a <ST_CurrentSystemTimeInfo>
PROPERTY CurrentTime : REFERENCE TO ST_CurrentSystemTimeInfo
GET
CurrentTime REF= _currentSystemTimeInfo;
END_GET
END_PROPERTY

// Sets the system time. Returns TRUE when done.
METHOD SetSystemTime : BOOL
VAR_INPUT
	timeToSet	: Tc2_Utilities.TIMESTRUCT;
END_VAR

VAR_OUTPUT
	error	: BOOL;	// Will be TRUE if an error occurs
	errorId	: TcError.AdsErrorCodes;	// Error code is reported here
END_VAR

VAR_INST
	setLocalTime	: Tc2_Utilities.NT_SetLocalTime :=(
		NETID := '',
		TMOUT := Tc2_System.DEFAULT_ADS_TIMEOUT);
END_VAR
setLocalTime(
	START := NOT setLocalTime.BUSY, 
	TIMESTR := timeToSet,
	ERR => error);
	
errorId := TcError.ToAdsErrorCode(TcError.ToAdsErrorCode(setLocalTime.ERRID));
SetSystemTime := NOT setLocalTime.BUSY;
END_METHOD

END_FUNCTION_BLOCK

// SOURCE/Time/I_LocalSystemTimeProvider
INTERFACE I_LocalSystemTimeProvider

METHOD PUBLIC ConvertToString : I_DateTimeToStringConverter
VAR_INPUT
END_VAR
END_METHOD

{attribute 'monitoring':='call'}
// Gets current system timo info as a <ST_CurrentSystemTimeInfo>
PROPERTY CurrentTime : REFERENCE TO ST_CurrentSystemTimeInfo
GET
END_GET
END_PROPERTY

END_INTERFACE

// TESTS/Test suites/Time/FB_LocalSystemTime_Tests
FUNCTION_BLOCK INTERNAL FB_LocalSystemTime_Tests EXTENDS TcUnit.FB_TestSuite
VAR_INPUT
END_VAR
VAR_OUTPUT
END_VAR
VAR
	_localSystemTimeProvider	: FB_LocalSystemTimeProvider;
END_VAR

_localSystemTimeProvider();
Test01_CheckSystemTime_ExpectValue();
Test02_SetSystemTime_ExpectNoErrorAndCorrectTimeRead();

METHOD Test01_CheckSystemTime_ExpectValue
VAR_INPUT
END_VAR

VAR
	emptyTimeStruct	: Tc2_Utilities.TIMESTRUCT;
END_VAR

IF TcUnit.TEST_ORDERED('Test01_CheckSystemTime_ExpectValue') THEN
	IF _localSystemTimeProvider.CurrentTime.IsValid THEN
		AssertTrue(
			Tc2_System.MEMCMP(ADR(emptyTimeStruct),
				ADR(_localSystemTimeProvider.CurrentTime.Value), 
				SIZEOF(Tc2_Utilities.TIMESTRUCT)) <> E_MemCmpResults.IDENTICAL,
			'System time returned an empty property value!');
		TcUnit.TEST_FINISHED();		
	END_IF
END_IF
END_METHOD

METHOD PRIVATE Test02_SetSystemTime_ExpectNoErrorAndCorrectTimeRead
VAR_INPUT
END_VAR
VAR CONSTANT
	timeToSet	: Tc2_Utilities.TIMESTRUCT := (
		wYear := 2026, 
		wMonth := 2, 
		wDay := 3, 
		wHour := 4,
		wMinute := 5,
		wSecond := 5,
		wMilliseconds := 7);
END_VAR
VAR
	error	: BOOL;
	errorId	: TcError.AdsErrorCodes;
END_VAR
VAR_INST
	testAssertionsDone_WaitForSystemTimeToBeSetBackToOriginalValue	: BOOL;
	originalTime	: Tc2_Utilities.TIMESTRUCT;
	timeSettingDone		: BOOL;
	waitForSynchronisationOfLocalSystemTime		: Tc2_Standard.TON := (PT := T#1200MS);
END_VAR
IF TcUnit.TEST_ORDERED('Test02_SetSystemTime_ExpectNoErrorAndCorrectTimeRead') THEN
	IF _localSystemTimeProvider.CurrentTime.IsValid THEN
		// Save original time to reset due to TwinCAT licensing system
		IF originalTime.wYear = 0 THEN
			originalTime := _localSystemTimeProvider.CurrentTime.Value;			
		END_IF
		
		// Set time only once
		IF NOT timeSettingDone AND_THEN _localSystemTimeProvider.SetSystemTime(timeToSet, error => error, errorId => errorId ) THEN
			waitForSynchronisationOfLocalSystemTime.IN := TRUE;
			AssertFalse(error, 
				'Error occured attempting to set system time');
			AssertTrue(errorId = TcError.AdsErrorCodes.ERR_NOERROR, 
				CONCAT('Error has occured - ', TO_STRING(errorId)));
			timeSettingDone := TRUE;				
		END_IF
		
		waitForSynchronisationOfLocalSystemTime(IN := timeSettingDone);
		// Since dwCycle minimum setting is 1 second (DWORD, seconds), we need to wait before we have a valid time value
		
		IF waitForSynchronisationOfLocalSystemTime.Q AND NOT 
			testAssertionsDone_WaitForSystemTimeToBeSetBackToOriginalValue 
		THEN
			AssertEquals_WORD(_localSystemTimeProvider.CurrentTime.Value.wYear, 2026, 'Year was not set correctly!');
			AssertEquals_WORD(_localSystemTimeProvider.CurrentTime.Value.wMonth, 2, 'Month was not set correctly!');
			AssertEquals_WORD(_localSystemTimeProvider.CurrentTime.Value.wDay, 3, 'Day was not set correctly!');
			AssertEquals_WORD(_localSystemTimeProvider.CurrentTime.Value.wHour, 4, 'Hour was not set correctly!');
			AssertEquals_WORD(_localSystemTimeProvider.CurrentTime.Value.wMinute, 5, 'Minute was not set correctly!');
			// Since synchronisation is done with 1 second (minimum), check the value range for second and millisecond
			AssertTrue(_localSystemTimeProvider.CurrentTime.Value.wSecond >= 6, 'Second was not set correctly!');
			AssertTrue(_localSystemTimeProvider.CurrentTime.Value.wMilliseconds >= 7, 'Millisecond was not set correctly!');
			testAssertionsDone_WaitForSystemTimeToBeSetBackToOriginalValue := TRUE;
		END_IF
		
		// Set time back othewise TwinCAT stops working due to invalid license :)
		IF testAssertionsDone_WaitForSystemTimeToBeSetBackToOriginalValue THEN
			IF _localSystemTimeProvider.SetSystemTime(originalTime) THEN
				TcUnit.TEST_FINISHED();	
			END_IF
		END_IF
	END_IF
END_IF
END_METHOD

END_FUNCTION_BLOCK

// TESTS/Test suites/FB_AdsHelper_Tests
// Subject under test
FUNCTION_BLOCK INTERNAL FB_AdsHelper_Tests EXTENDS FB_TestSuite

// Create instance variables that will be accesible for all tests
VAR
END_VAR

// Call your test methods here
Test_NetIdToString_AllZeros_ExpectEmptyString();
Test_MasterAddress();

METHOD Test_MasterAddress

VAR_INST
	masterNetId	: Tc2_System.T_AmsNetID := '0.0.0.0.0.5';
END_VAR
TcUnit.TEST('Test_MasterAddress');

AssertEquals_DINT(
	Expected := 24,
	Actual := 24,
	Message := 'Getting address from master netId was incorrect!');
	
TcUnit.TEST_FINISHED();
END_METHOD

METHOD PRIVATE Test_NetIdToString_AllZeros_ExpectEmptyString

(* Instanced variables are VERY useful for writing tests since tests are run in paralel (by default).
By instantiating local variables that are not placed on the same stack as method (values are retained between calls)
you make sure that the SUT is not changed by some other test. *)
VAR_INST
	
END_VAR

// Place temporary variables here
VAR
	emptyNetId	: Tc2_System.T_AmsNetIdArr;
END_VAR
// The name of the test, is the same as method name!
TcUnit.TEST('Test_NetIdToString_AllZeros_ExpectEmptyString');

// Do your assertions here...
AssertEquals_STRING(
	Expected := '',
	Actual := AdsHelper.NetIdToString(emptyNetId),
	Message := 'An empty netId should return an empty string!');

TcUnit.TEST_FINISHED();
END_METHOD

END_FUNCTION_BLOCK

// TESTS/Test suites/FB_ArrayHelper_Tests
FUNCTION_BLOCK INTERNAL FB_ArrayHelper_Tests EXTENDS FB_TestSuite
VAR_INPUT
END_VAR
VAR_OUTPUT
END_VAR

Test01_GetArrayElementCount();
Test02_GetArrayMaxIndex();
Test03_InsertNumber();
Test04_InsertString();
Test05_InsertStruct();
Test06_ShiftUp_ExpectLastElementOverwriteFirstElementZero();
Test07_SetAtFirstEmptySlot();
Test08_AllMethods_provideNonArrayVar_ExpectNothing();
Test09_InsertIntoEmptyArray_ExpectOnlyFirstItem();
Test10_CheckIfArrayContainsItem();
Test11_ClearArray_ExpectEmptyArray();
Test12_ReferenceToArrayWithAllMethods_ExpectNormalResults();
Test13_FindLastOccupiedItem();
Test14_ShiftDown_ExpectFirstElementOverwriteLastElementZero();

METHOD Test01_GetArrayElementCount
VAR_INPUT
END_VAR
VAR
	arr		: ARRAY[0..99] OF REAL;
	arr2	: ARRAY[22..33] OF REAL;
END_VAR
TcUnit.TEST('Test01_GetArrayElementCount');

AssertEquals_DINT(
	Actual := ArrayHelper.GetElementCount(arr := arr, dataType := arr[0]),
	Expected := 100,
	Message := 'Getting array element count failed!');
	
AssertEquals_DINT(
	Actual := ArrayHelper.GetElementCount(arr := arr2, dataType := arr2[22]),
	Expected := 33 - 22 + 1,
	Message := 'Getting array element count for array with non-zero start element index failed!');
	
TcUnit.TEST_FINISHED();
END_METHOD

METHOD Test02_GetArrayMaxIndex
VAR_INPUT
END_VAR
VAR
	arr		: ARRAY[0..99] OF REAL;
	arr2	: ARRAY[22..33] OF REAL;
END_VAR
TcUnit.TEST('Test02_GetArrayMaxIndex');

AssertEquals_DINT(
	Actual := ArrayHelper.GetMaxIndex(arr := arr, dataType := arr[0], startIndex := 0),
	Expected := 99,
	Message := 'Getting array maximum index failed!');
	
AssertEquals_DINT(
	Actual := ArrayHelper.GetMaxIndex(arr := arr2, dataType := arr2[22], startIndex := 22),
	Expected := 33,
	Message := 'Getting array maximum index for array with non-zero start element index failed!');
	
TcUnit.TEST_FINISHED();
END_METHOD

METHOD PRIVATE Test03_InsertNumber
VAR_INPUT
END_VAR

VAR
	i		: INT;
	value	: INT := 99;
	arr		: ARRAY [0..10] OF INT;
END_VAR
TcUnit.TEST('Test03_InsertNumber');

FOR i := 0 TO 10 BY 1 DO
	arr[i] := i;
END_FOR

ArrayHelper.InsertAtStart(
	arr := arr,
	item := value);
	
AssertEquals_INT(
	Expected := value,
	Actual := arr[0],
	Message := 'First item was not inserted properly!');
	
AssertEquals_INT(
	Expected := 9,
	Actual := arr[10],
	Message := 'Last item was not removed from the array!!');
	
TcUnit.TEST_FINISHED();
END_METHOD

METHOD PRIVATE Test04_InsertString
VAR_INPUT
END_VAR

VAR
	i		: INT;
	value	: STRING := '9';
	arr		: ARRAY [0..10] OF STRING;
END_VAR
TcUnit.TEST('Test04_InsertString');

FOR i := 0 TO 10 BY 1 DO
	arr[i] := INT_TO_STRING(i);
END_FOR

ArrayHelper.InsertAtStart(
	arr := arr,
	item := value);
	
AssertEquals_STRING(
 	Actual:= arr[0],
	Expected := value,
	Message := 'First item was not inserted properly!');
	
AssertEquals_STRING(
	Expected := '9',
	Actual := arr[10],
	Message := 'Last item was not removed from the array!!');
	
TcUnit.TEST_FINISHED();
END_METHOD

METHOD Test05_InsertStruct

VAR
	i		: INT;
	value	: ST_GenericError;
	arr		: ARRAY [0..10] OF ST_GenericError;
END_VAR
TcUnit.TEST('Test05_InsertStruct');

FOR i := 0 TO 10 BY 1 DO
	arr[i].Code := i;
	arr[i].Message := INT_TO_STRING(i);
END_FOR

ArrayHelper.InsertAtStart(
	arr := arr,
	item := value);
	
AssertEquals(
	Expected := value,
	Actual := arr[0],
	Message := 'First item was not inserted properly!');
	
AssertEquals_STRING(
	Expected := '9',
	Actual := arr[10].Message,
	Message := 'Last item was not removed from the array!');
	
AssertEquals_STRING(
	Expected := '9',
	Actual := arr[10].Message,
	Message := 'Last item was not removed from the array!');
	
TcUnit.TEST_FINISHED();
END_METHOD

METHOD Test06_ShiftUp_ExpectLastElementOverwriteFirstElementZero
VAR_INPUT
END_VAR

VAR_INST
	arr	: ARRAY[0..20] OF INT;
	i	: int;
END_VAR
TcUnit.TEST('Test06_ShiftUp_ExpectLastElementOverwriteFirstElementZero');

FOR i := 0 TO 20 BY 1 DO
	arr[i] := i;
END_FOR

ArrayHelper.ShiftUp(
	arr := arr,
	dataType := arr[0]);
AssertEquals_INT(
	Actual := arr[0],
	Expected := 0,
	Message := 'Shifting the array up, first element should be set to 0!');
	
FOR i := 1 TO 20 BY 1 DO
	AssertEquals_INT(
		Actual := arr[i],
		Expected := i-1,
		Message := Tc2_Standard.CONCAT('Shifting up failed! Incorrect value at position ', TO_STRING(i)));
END_FOR
	
TcUnit.TEST_FINISHED();
END_METHOD

METHOD Test07_SetAtFirstEmptySlot
VAR_INPUT
END_VAR

VAR
	arr		: ARRAY[0..69] OF T_ArrayIndexer;
	arr2	: ARRAY[0..69] OF BOOL;
	valueToSet	: T_ArrayIndexer := 9999;
	i	: T_ArrayIndexer;
	boolValueToSet	: BOOL := TRUE;
END_VAR
TcUnit.TEST('Test07_SetAtFirstEmptySlot');

FOR i := 0 TO 30 BY 1 DO
	arr[i] := i + 1;
	arr2[i] := TRUE;
END_FOR

ArrayHelper.SetAtFirstEmptySlot(
	arr := arr,
	item := valueToSet);

ArrayHelper.SetAtFirstEmptySlot(
	arr := arr2,
	item := boolValueToSet);

FOR i := 0 TO 30 BY 1 DO
	AssertEquals_DINT(
		Expected := i + 1,
		Actual := arr[i],
		Message := 'Setting first empty slot should not have changed non-empty fields!');
		
	AssertTrue(
		Condition := arr2[i],
		Message := 'Setting first empty slot for array of booleans should not have changed non-empty fields!');
END_FOR

AssertEquals(
	Expected := valueToSet,
	Actual := arr[31],
	Message := 'Setting first empty slot failed, first empty element differs!');
	
AssertTrue(
	Condition := arr2[31],
	Message := 'Setting first empty slot failed, first empty element should be set to TRUE!');
	
AssertEquals_DINT(
	Expected := 0,
	Actual := arr[32],
	Message := 'Setting first empty slot failed, item after the inserted slot should be empty!');
	
AssertFalse(
	Condition := arr2[32],
	Message := 'Setting first empty slot failed, item after the inserted slot should be empty!');	
	

TcUnit.TEST_FINISHED();
END_METHOD

METHOD Test08_AllMethods_provideNonArrayVar_ExpectNothing
VAR_INPUT
END_VAR
VAR
	notAnArray	: BOOL := TRUE;
	val			: BOOL;
END_VAR
TcUnit.TEST('Tes08_AllMethods_provideNonArrayVar_ExpectNothing');

ArrayHelper.GetElementCount(arr := notAnArray, dataType := val);
AssertTrue(
	Condition := notAnArray, 
	Message := 'When non-array is provided to any method, the method should not execute anything!');

AssertEquals_DINT(
	Actual := ArrayHelper.GetMaxIndex(arr := notAnArray, dataType := val, startIndex := 0),
	Expected := 0,
	Message := 'When non-array is provided, max index returned should be 0!');
	
AssertTrue(
	Condition := notAnArray, 
	Message := 'When non-array is provided to any method, the method should not execute anything!');

	
TcUnit.TEST_FINISHED();
END_METHOD

METHOD Test09_InsertIntoEmptyArray_ExpectOnlyFirstItem
VAR_INPUT
END_VAR

VAR_INST
	arr			: ARRAY[0..20] OF ST_GenericError;
	item		: ST_GenericError := (Code := 0, Message := '0');
	emptyItem	: ST_GenericError;
	i 			: T_ArrayIndexer;
END_VAR
TcUnit.TEST('Test09_InsertIntoEmptyArray_ExpectOnlyFirstItem');

FOR i := 0 TO 20 BY 1 DO
	AssertEquals(Actual := arr[i], Expected := emptyItem, Message := 'Wrong array initialization!');
END_FOR

ArrayHelper.InsertAtStart(arr := arr, item := item);

AssertEquals(
	Actual := arr[0], 
	Expected := item, 
	Message := 'InsertAtStart should have first item in array the same as item being inserted!');
	
FOR i := 1 TO 20 BY 1 DO
	AssertEquals(Actual := arr[i], Expected := emptyItem, 
		Message := Tc2_Standard.CONCAT(
			STR1 := 'InsertAtStart should have left other elements unchanged! Changed element at index ', 
			STR2 := TO_STRING(i) ));
END_FOR

ArrayHelper.InsertAtStart(arr := arr, item := item);
AssertEquals(
	Actual := arr[0], 
	Expected := item, 
	Message := 'Inserting at start for the second time - 1st item is incorrect!');
AssertEquals(
	Actual := arr[1], 
	Expected := item, 
	Message := 'Inserting at start for the second time - 2nd item is incorrect!');	

TcUnit.TEST_FINISHED();
END_METHOD

METHOD Test10_CheckIfArrayContainsItem
VAR_INST
	arr		: ARRAY[0..10] OF STRING;
	item	: STRING := 'mwah';
END_VAR
TcUnit.TEST('Test10_CheckIfArrayContainsItem');

ArrayHelper.Clear(arr);
AssertFalse(
	Condition := ArrayHelper.DoesArrayContainItem(arr, item),
	Message := 'Array does not contain the item, method should return FALSE.');

arr[0] := item;

AssertTrue(
	Condition := ArrayHelper.DoesArrayContainItem(arr, item),
	Message := 'Array does contain the item on 0th index, method should return TRUE.');
	
arr[0] := '';
arr[5] := item;

AssertTrue(
	Condition := ArrayHelper.DoesArrayContainItem(arr, item),
	Message := 'Array does contain the item on 5th index, method should return TRUE.');
	
arr[5] := '';
arr[10] := item;	
AssertTrue(
	Condition := ArrayHelper.DoesArrayContainItem(arr, item),
	Message := 'Array does contain the item on 10th index, method should return TRUE.');

arr[0] := 'lalala';
arr[3] := 'aahah';
AssertTrue(
	Condition := ArrayHelper.DoesArrayContainItem(arr, item),
	Message := 'Array does contain the item on 10th index, but also includes non empty elements before, method should return TRUE.');

arr[2] := item;
AssertTrue(
	Condition := ArrayHelper.DoesArrayContainItem(arr, item),
	Message := 'Array does contain the item on 2nd index, but also includes non empty elements before and after, method should return TRUE.');	
	
TcUnit.TEST_FINISHED();
END_METHOD

METHOD Test11_ClearArray_ExpectEmptyArray
VAR_INPUT
END_VAR
VAR_INST
	arrUnmodified	: ARRAY[0..20] OF BOOL;
	arrModified		: ARRAY[0..20] OF BOOL;
	idx				: T_ArrayIndexer;
END_VAR
TcUnit.TEST('Test11_ClearArray_ExpectEmptyArray');

FOR idx := 0 TO 20 BY 1 DO
	arrModified[idx] := TRUE;
END_FOR

AssertTrue(
	Condition := ArrayHelper.Clear(arrModified),
	Message := 'Clearing array returned FALSE when it should have been TRUE.');

AssertArrayEquals_BOOL(
	Actuals := arrModified,
	Expecteds := arrUnmodified,
	Message := 'Array contents were not cleared.');

TcUnit.TEST_FINISHED();
END_METHOD

METHOD Test12_ReferenceToArrayWithAllMethods_ExpectNormalResults
VAR_INST
	arr			: ARRAY[0..10] OF REAL;
	refArr		: REFERENCE TO ARRAY[0..10] OF REAL;
	arrEmpty	: ARRAY[0..10] OF REAL;
	findResult	: REAL;
END_VAR
TcUnit.TEST('Test12_ReferenceToArrayWithAllMethods_ExpectNormalResults');
refarr REF= arr;
arr[5] := 22.2;

ArrayHelper.Clear(refArr);
AssertArrayEquals_REAL(
	Actuals := arr,
	Expecteds := arrEmpty,
	Delta := 0,
	Message := 'Clear array failed.');
	
arr[6] := 5.3;
AssertTrue(
	Condition := ArrayHelper.DoesArrayContainItem(arr := refArr, item := arr[6]),
	Message := 'DoesArrayContainItem failed.');

AssertTrue(
	Condition := ArrayHelper.FindLastOccupiedItem(refArr, refArr[0], findResult),
	Message := 'FindLastOccupiedItem failed (returned FALSE).');

AssertEquals_REAL(
	Actual := findResult,
	Expected := 5.3,
	Delta := 0,
	Message := 'FindLastOccupiedItem output value was incorrect.');
	
AssertEquals_DINT(
	Actual := ArrayHelper.GetElementCount(refArr, refArr[0]),
	Expected := 11,
	Message := 'GetEleeentCount failed.');
	
AssertEquals_DINT(
	Actual := ArrayHelper.GetMaxIndex(refArr, refArr[0], 0),
	Expected := 10,
	Message := 'GetMaxIndex failed.');
	
ArrayHelper.InsertAtStart(refArr, findResult);
AssertEquals_REAL(
	Actual := refArr[0],
	Expected := 5.3,
	Delta := 0.0,
	Message := 'InsertAtStart failed');

arr[0] := 0;	
ArrayHelper.SetAtFirstEmptySlot(refArr, findResult);	
AssertEquals(
	Expected := findResult,
	Actual := refArr[0],
	Message := 'SetAtFirstEmptySlot failed.');
	
arr[1] := 5.5;
ArrayHelper.ShiftDown(refArr, refArr[0]);
AssertEquals_REAL(
	Actual := refArr[0],
	Expected := 5.5,
	Delta := 0.0,
	Message := 'ShiftDown failed.');

ArrayHelper.ShiftUp(refARr, refArr[0]);
AssertEquals_REAL(
	Actual := refArr[1],
	Expected := 5.5,
	Delta := 0.0,
	Message := 'ShiftUp failed.');

TcUnit.TEST_FINISHED();
END_METHOD

METHOD Test13_FindLastOccupiedItem
VAR_INPUT
END_VAR

VAR_INST
	arr	: ARRAY[0..10] OF INT;
	result	: int;
END_VAR
TcUnit.TEST('Test13_FindLastOccupiedItem');

AssertFalse(
	Condition := ArrayHelper.FindLastOccupiedItem(arr, arr[0], result),
	Message := 'Empty array should return FALSE.');
	
arr[5] := 5;

AssertTrue(	
	Condition := ArrayHelper.FindLastOccupiedItem(arr, arr[0], result),
	Message := 'Expected TRUE, 5th element is not empty.');
	
AssertEquals_INT(
	Actual := result,
	Expected := 5,
	Message := 'Incorrect result when finding last occupied element.');
	
TcUnit.TEST_FINISHED();
END_METHOD

METHOD Test14_ShiftDown_ExpectFirstElementOverwriteLastElementZero
VAR_INPUT
END_VAR

VAR
	arr	: ARRAY[0..20] OF INT;
	i	: int;
END_VAR
TcUnit.TEST('Test14_ShiftDown_ExpectFirstElementOverwriteLastElementZero');

FOR i := 0 TO 20 BY 1 DO
	arr[i] := i;
END_FOR

ArrayHelper.ShiftDown(
	arr := arr,
	dataType := arr[0]);
	
AssertEquals_INT(
	Actual := arr[20],
	Expected := 0,
	Message := 'Shifting the array down, last element should be set to 0!');
	
FOR i := 19 TO 0 BY -1 DO
	AssertEquals_INT(
		Actual := arr[i],
		Expected := i+1,
		Message := Tc2_Standard.CONCAT('Shifting up failed! Incorrect value at position ', TO_STRING(i)));
END_FOR
	
TcUnit.TEST_FINISHED();
END_METHOD

END_FUNCTION_BLOCK

// TESTS/Test suites/FB_BoolEx_Tests
FUNCTION_BLOCK INTERNAL FB_BoolEx_Tests EXTENDS FB_TestSuite
VAR_INPUT
END_VAR
VAR_OUTPUT
END_VAR
VAR
	_boolVariable	: BOOL;
	_intVariable	: INT;
	_boolEx			: BoolEx := (variable := _boolVariable);
END_VAR

Test01_BooleanTrue_ExpectTrueAfterElapsedTime();
Test02_BooleanFalse_ExpectTrueAfterElapsedTime();
Test03_RisingAndFallingEdge_ExpectPulses();
Test04_GetAndSetValue();
Test05_Toggle_ExpectValueInverts();
Test06_PulseWithInterval_100ms_ExpectValueChangeEvery100ms();
Test07_Set_ExpectTrue();
Test08_Reset_ExpectFalse();

METHOD Test01_BooleanTrue_ExpectTrueAfterElapsedTime
VAR_INPUT
		
